FUNCTION_BLOCK FB_FanucRobot_Basic IMPLEMENTS IBasicElement
VAR_INPUT
    Estop  : BOOL; // PLC ->send to Robot E-Stop
    OpMode : E_FanucRobotOpMode := RSR01; // Select Fanuc robot prog RSR1~RSR3
    Start  : BOOL;
    Reset  : BOOL; // Reset Fanuc Robot prog
    Hold   : BOOL; // PLC - > Robot send hold command
	ManualCtrl : REFERENCE TO ST_Manual_FanucRobot;
END_VAR

VAR_OUTPUT
    qEnable       : BOOL;
    qFault        : BOOL;
    E_Stop_Output : BOOL; // Touch pannel's E-Stop has been trig;
    Halt          : BOOL; // True : Robot in helt state.
    Error         : BOOL; // True : Robot has error
    ErrorID       : UDINT; // Error ID output
	ErrMsg 		  : T_MaxString;	  
END_VAR

VAR
    // Slot1
    _rawIn_UI AT %I*  : ARRAY[0..3] OF BYTE; // UI : Fanuc robot default input rawdate
    _rawOut_UO AT %Q* : ARRAY[0..3] OF BYTE; // UO : Fanuc robot default output rawdate
    // Slot2
    _rawIn_DI AT %I*           : ARRAY[0..31] OF BYTE; // DI : user define input rawdate
    _rawOut_DO AT %Q*          : ARRAY[0..31] OF BYTE; // DO : user define output rawdate
    _EIPConnectionState AT %I* : UINT; // EIP connection State (EL6652 to Fanuc Robot)
    _FanucEIPState AT %I*      : UINT; // EIP module links to FanucRobot state
    _UI1                       : ST_FanucUI1; // Fanuc Robot default Input
    _UO1                       : ST_FanucUO1; // Fanuc Robot default Output
    _DO1                       : ST_Fanuc_WarehouseHandshake; // Fanuc robot program's handshake for clampA warehouse pick / place box
    _DO2                       : ST_Fanuc_WarehouseHandshake; // Fanuc robot program's handshake for clampB warehouse pick / place box
    _DO3                       : ST_Fanuc_AbsMove; // Fanuc robot program's handshake for clampA to target area pick / place box
    _DO4                       : ST_Fanuc_AbsMove; // Fanuc robot program's handshake for clampB to target area pick / place box
    _DO5                       : ST_Fanuc_GeneralCommand; // Fanuc robot program's handshake for general control
    _DO6                       : ST_ReadWriteParaCmd; // Fanuc robot Read/Write parameter command 
    _DO7                       : INT; // Write process X position offset
    _DO8                       : INT; // Write process Y position offset
    _DO9                       : INT; // Write process Z position offset
    _DO10                      : INT; // Write process W position offset
    _DO11                      : INT; // Write process P position offset
    _DO12                      : INT; // Write process R position offset
    _Do13                      : INT; // Write process Area index
    _Do14                      : INT; // Write process Address index
    _Do15                      : INT; // Write process Layer index
    _DO16                      : INT; // Write process Slide index
    _DO17                      : ST_CCD_ZoneUse; // Set Robot use ccd or not.
    _DI1                       : ST_Fanuc_Status; // Fanuc robot program's handshake for process status
    _DI2                       : INT; // Readprocess X position offset
    _DI3                       : INT; // Read process Y position offset
    _DI4                       : INT; // Read process Z position offset
    _DI5                       : INT; // Read process W position offset
    _DI6                       : INT; // Read process P position offset
    _DI7                       : INT; // Read process R position offset
    _DI8                       : INT; // Read process Area index
    _DI9                       : INT; // Read process Address index
    _DI10                      : INT; // Read Process Layer index
    _DI11                      : INT; // Read Process Slide index
    _DI12                      : ST_ReadWriteParaStatus; // Read/Write process Status
    _VelocityCommand           : ST_IntToBool; // Robot coordenate velocity
    // Prog inside
    eState               : E_MethodStatus_Basic;
    uiRobotExecutingStep : UINT;
    uiRobotResettingStep : UINT;
    _Error               : BOOL;
    _Abort               : BOOL;
    TON_Restart_delay    : TON;
    TON_Reset_delay      : TON;
    Rtrig_RebootRobot    : R_TRIG;
    //fbReadSingleOffsetData  : FB_ReadSingleOffsetData;
    //fbWriteSingleOffsetData : FB_WriteSingleOffsetData;
    _Status               : T_MaxString;
    _eOpMode              : E_FanucRobotOpMode;
    _ModeChanging         : BOOL;
    _Completed            : BOOL;
    _ModeChanged          : BOOL;
    _uiRSR01_Step         : UINT;
    _uiRSR02_Step         : UINT;
    _uiRSR03_Step         : UINT;
    _RetryCount           : INT := 0;
    Ton_SetProgTimeOut    : TON; // This timer is used to counting the time to switch FanucRobot prog over range.
    _RSR1_Ready           : BOOL; // Fanuc Robot running in RSR1 prog, allow to Warehouse or AbsMove command.
    _RSR2_Completed       : BOOL; // Fanuc Robot finished the homing prog.
    _RSR3_Ready           : BOOL; // Fanuc Robot ready to work.
    TON_ResetFixDelay     : TON;
    Ton_RSR_SwitchDelay   : TON; // This timer is used to counting the time to switch rsr prog
    ErrorCode             : ST_IntToBool; // This value is which read from fanuc robot.
    Ton_START_SwitchDelay : TON; // This timer is used to counting the time to switch Start signal, Fanuc process need on 0.3s and off
END_VAR

VAR CONSTANT
    RetryMaxTimes   : INT  := 3;
    tSwitchProgTime : TIME := T#1S;
    tResetFixTime   : TIME := T#0.3S;
END_VAR

// Active base units.
A00_BaseUnit();
// Active mode controller
A10_ModeControl();
// Active state controller
A20_ErrorHandle();

Update();

ACTION A00_BaseUnit:
Ton_SetProgTimeOut(PT := tSwitchProgTime);
TON_Restart_delay(PT := T#1S); // Fanuc Robot need IMSTP on over 1s
TON_Reset_delay(PT := T#1S);
TON_ResetFixDelay(PT := tResetFixTime);
Ton_RSR_SwitchDelay(PT := T#0.3S);
Ton_START_SwitchDelay(PT := T#0.4S); // Fanuc Robot need on 0.3s and then set off
E_Stop_Output := _DI12.E_Stop;
END_ACTION

ACTION A10_ModeControl:
CASE _eOpMode OF
	E_FanucRobotOpMode.RSR01:
		M_ControlRSR01(bCompleted=> _Completed, ModeChanging=> _ModeChanging, ModeChanged=> _ModeChanged);
	E_FanucRobotOpMode.RSR02:
		M_ControlRSR02(bCompleted=> _Completed, ModeChanging=> _ModeChanging, ModeChanged=> _ModeChanged);
END_CASE
END_ACTION

ACTION A20_ErrorHandle:
ErrMsg := _Status;
END_ACTION

ACTION A20_StateControl:
TON_Restart_delay(PT := T#0.5S);
TON_Reset_delay(PT:=T#0.5S);
CASE eState OF
    E_MethodStatus_Basic.STATE_DORMANT:
        Enable(FALSE);
        M_Reset(FALSE);
        uiRobotExecutingStep := 0;
        uiRobotResettingStep := 0;

		IF _eOpMode = RSR01 OR _eOpMode = RSR02 OR _eOpMode = RSR03 THEN
			eState := E_MethodStatus_Basic.STATE_EXECUTING;
		END_IF
    E_MethodStatus_Basic.STATE_EXECUTING:
        CASE uiRobotExecutingStep OF
            0:
                Enable(iTrigger := TRUE);
                M_Reset(iTrigger := TRUE);
				TON_Reset_delay.in := TRUE;
                IF TON_Reset_delay.Q THEN
                    uiRobotExecutingStep := 100;
                END_IF
            100:
                M_Reset(iTrigger := FALSE);
				TON_Reset_delay.IN := FALSE;
                IF _UO1.UO01_CmdEnabled AND _UO1.UO02_SystemReady THEN
					_VelocityCommand.nInt := 1;
                    uiRobotExecutingStep := 200;
                END_IF
            200:
				// Clear Fanuc robot's action
				GVL_ADS.AutoMode_WarehouseMotoWithRobotMove.HandShake.Execute := FALSE;
				GVL_ADS.AutoMode_RobotAbsMove.HandShake.Execute := FALSE;
				_DO1.bExecute := FALSE; // Warehouse with robot clampA
				_DO2.bExecute := FALSE; // Warehouse with robot clampB
				_DO3.bExecute := FALSE; // AbsMove with robot clampA
				_DO4.bExecute := FALSE; // AbsMove with robot clampB
				uiRobotExecutingStep := 250;
			300:
				// Switch RSR3 and read all of offset data
				GVL_ADS.FanucRobot_ReadAllOffsetData.Command.Execute := TRUE;
				IF GVL_ADS.FanucRobot_ReadAllOffsetData.Status.Done THEN
					uiRobotExecutingStep := 400;
				ELSIF GVL_ADS.FanucRobot_ReadAllOffsetData.Status.Error THEN
					_Error := TRUE;
					_Status := 'Read All offset data failue';
				END_IF
			400:
                _UI1.UI09_RSR1 := TRUE;

                IF _UO1.UO11_ACK1 THEN
                    uiRobotExecutingStep := 500;
                END_IF
            500:
                _UI1.UI09_RSR1       := FALSE;
				_VelocityCommand.nInt := 30;
                uiRobotExecutingStep := 600;
            600: // Wait command
				_DO5.ClampA_Close :=  GVL_ADS.FanucRobot_General.Command.ClampA_Close;
				_DO5.ClampA_Open := GVL_ADS.FanucRobot_General.Command.ClampA_Open;
				_DO5.ClampB_Close := GVL_ADS.FanucRobot_General.Command.ClampB_Close;
				_DO5.ClampB_Open := GVL_ADS.FanucRobot_General.Command.ClampB_Open;
				_DO6.ByPassClampSensor := GVL_ADS.FanucRobot_General.Command.ByPassClampSensor;
				GVL_ADS.FanucRobot_General.Status.ClampA_Open := _DI1.ClampA_Open;
				GVL_ADS.FanucRobot_General.Status.ClampA_Sensor := _DI1.ClampA_Sensor;
				GVL_ADS.FanucRobot_General.Status.ClampB_Open := _DI1.ClampB_Open ;
				GVL_ADS.FanucRobot_General.Status.ClampB_Sensor := _DI1.ClampB_Sensor;
				_VelocityCommand.nInt := GVL_ADS.FanucRobot_General.Command.RobotVelocity;
        END_CASE

        IF (*qFault OR *)_Error THEN
            //Soft E-Stop will cause Fault error
            eState := E_MethodStatus_Basic.STATE_ERROR;
        ELSIF _Abort THEN
            eState := E_MethodStatus_Basic.STATE_ABORTING;
		ELSIF Estop THEN
			eState := E_MethodStatus_Basic.STATE_ABORTING;
        END_IF
    E_MethodStatus_Basic.STATE_DONE:
        ;
    E_MethodStatus_Basic.STATE_ABORTING:
	;
//        Hold();

        IF _UO1.UO04_PrgPaused THEN
            eState := E_MethodStatus_Basic.STATE_Aborted;
        END_IF
    E_MethodStatus_Basic.STATE_Aborted:
        IF _UI1.UI05_FaultReset OR GVL.Reset THEN
            eState := E_MethodStatus_Basic.STATE_RESETTING;
        END_IF
    E_MethodStatus_Basic.STATE_ERROR:
        IF _UI1.UI05_FaultReset THEN
            eState := E_MethodStatus_Basic.STATE_RESETTING;
        END_IF
    E_MethodStatus_Basic.STATE_RESETTING:
        CASE uiRobotResettingStep OF
            0:
                IF NOT _UO1.UO06_Fault THEN
                    IF NOT _UO1.UO04_PrgPaused THEN
                        uiRobotResettingStep := 1000;
                    ELSE
                        uiRobotResettingStep := 2000;
                    END_IF
                ELSE
                    uiRobotResettingStep := 1000;
                END_IF
            1000:
                M_Reset(TRUE);
				TON_Reset_delay.in := TRUE;
				IF TON_Reset_delay.Q THEN
                	uiRobotResettingStep := 1010;
				END_IF
            1010:
				TON_Reset_delay.IN :=FALSE;
                M_Reset(FALSE);
                uiRobotResettingStep := 9000;
            2000:
                _UI1.UI02_Hold       := TRUE;
                TON_Restart_delay.IN := TRUE; // TimeCount start

                IF TON_Restart_delay.Q THEN
                    uiRobotResettingStep := 2100;
                END_IF
            2100:
                TON_Restart_delay.IN := FALSE;
                _UI1.UI06_Start      := TRUE;
                uiRobotResettingStep := 9000;
            9000:
                IF NOT qFault THEN
                    eState := E_MethodStatus_Basic.STATE_DORMANT;
                END_IF
        END_CASE
END_CASE
Rtrig_RebootRobot(CLK:= GVL.MachineReset.AllReset);
IF Rtrig_RebootRobot.Q	AND qFault THEN
	ReBoot();
END_IF
END_ACTION

PROPERTY AbsMoveClampA_Handshake : ST_Fanuc_AbsMove
GET
AbsMoveClampA_Handshake := _DO3;
END_GET
SET
// Outside -> FB 
_DO3 := AbsMoveClampA_Handshake;
END_SET
END_PROPERTY

PROPERTY AbsMoveClampB_Handshake : ST_Fanuc_AbsMove
GET
AbsMoveClampB_Handshake := _DO4;
END_GET
SET
// Outside -> FB 
_DO4 := AbsMoveClampB_Handshake;
END_SET
END_PROPERTY

PROPERTY Bzone_AllowWork : Bool
GET
Bzone_AllowWork := THIS^._DO6.Bzone_AllowWork;
END_GET
SET
 THIS^._DO6.Bzone_AllowWork :=Bzone_AllowWork ;
END_SET
END_PROPERTY

PROPERTY BZoneInWork : Bool
GET
BZoneInWork := THIS^._DI12.BzoneInWork;
END_GET
END_PROPERTY

PROPERTY Command : ST_FanucUO1
GET
Command := _UO1;
END_GET
SET
_UO1 := Command;
END_SET
END_PROPERTY

METHOD Enable : BOOL
VAR_INPUT
iTrigger:BOOL;
END_VAR
VAR
	_RobotEnable:BOOL;
END_VAR
_RobotEnable:=iTrigger (*AND NOT Fault()*);

_UI1.UI01_IMSP:=_RobotEnable;
_UI1.UI02_Hold:=_RobotEnable;
_UI1.UI03_SFSP:=_RobotEnable;
_UI1.UI08_Enable:=_RobotEnable;
END_METHOD

METHOD EStop
VAR_INPUT
END_VAR
_UI1.UI03_SFSP:=FALSE;
END_METHOD

PROPERTY FanucRobot_MotionStatus : ST_Fanuc_Status
GET
FanucRobot_MotionStatus := _DI1;
END_GET
END_PROPERTY

METHOD Fault : BOOL
VAR_INPUT
END_VAR
VAR_INST
	bConectionError : BOOL;
END_VAR
bConectionError := (_EIPConnectionState <>0) OR (_FanucEIPState <> 0);
Fault:=_UO1.UO06_Fault OR _UO1.UO09_BattAlarm OR _DI1.Error OR bConectionError OR _UO1.UO08_TPEnabled;
END_METHOD

METHOD GetModelState
VAR_INPUT
END_VAR
VAR_OUTPUT
    xDone : BOOL;
    xBusy : BOOL;
    xError : BOOL;
    xAborted : BOOL;
    iErrorID : UDINT;
	UniqueErrorCode : STRING;
END_VAR
xError := Error;
iErrorID := INT_TO_UDINT(ErrorCode.nInt);
END_METHOD

METHOD GetName : STRING
VAR_INPUT
END_VAR
GetName := 'Fanuc Robot';
END_METHOD

METHOD Hold
VAR_INPUT
END_VAR
_UI1.UI02_Hold:=FALSE;
END_METHOD

PROPERTY Homed : Bool
GET
Homed := _RSR2_Completed OR _UO1.UO07_AtPerch;
END_GET
END_PROPERTY

PROPERTY LayerIndex : INT
SET
_Do15 := LayerIndex;
END_SET
END_PROPERTY

METHOD M_ActiveRSR01
VAR_INPUT
END_VAR
VAR_OUTPUT
	bCompleted : BOOL;
END_VAR
CASE eState OF
    E_MethodStatus_Basic.STATE_DORMANT:
        Enable(FALSE);
        M_Reset(FALSE);
        _uiRSR01_Step        := 0;
        uiRobotExecutingStep := 0;
        uiRobotResettingStep := 0;
        _RSR1_Ready          := FALSE;
        _RSR2_Completed      := FALSE;
        _RSR3_Ready          := FALSE;
        TON_Reset_delay.IN   := FALSE;
        _RSR1_Ready          := FALSE;

        IF _eOpMode = RSR01 OR _eOpMode = RSR02 OR _eOpMode = RSR03 THEN
            eState := E_MethodStatus_Basic.STATE_EXECUTING;
        END_IF
    E_MethodStatus_Basic.STATE_EXECUTING:
        CASE uiRobotExecutingStep OF
            0:
                Enable(iTrigger := TRUE);
                TON_Restart_delay.IN := TRUE;

                IF TON_Restart_delay.Q THEN
                    uiRobotExecutingStep := 10;
                END_IF
            10:
                TON_Restart_delay.IN := FALSE;
                M_Reset(iTrigger := TRUE);
                _UI1.UI04_CycleStop  := TRUE;
                TON_ResetFixDelay.IN := TRUE;

                IF TON_ResetFixDelay.Q THEN
                    uiRobotExecutingStep := 100;
                END_IF
            100:
                TON_ResetFixDelay.IN := FALSE;
                TON_Reset_delay.in   := TRUE;
                M_Reset(iTrigger := FALSE);
                _UI1.UI04_CycleStop := FALSE;

                IF TON_Reset_delay.Q THEN
                    IF _UO1.UO01_CmdEnabled AND _UO1.UO02_SystemReady THEN
                        _Error                := FALSE;
						Enable(iTrigger := TRUE); // 20250428 Albert
                        _VelocityCommand.nInt := 1;
                        uiRobotExecutingStep  := 200;
                    ELSIF Error THEN
                        eState := E_MethodStatus_Basic.STATE_ERROR;
                    END_IF
                END_IF
            200:
                // Clear Fanuc robot's action
                TON_Reset_delay.IN                                            := FALSE;
                GVL_ADS.AutoMode_WarehouseMotoWithRobotMove.HandShake.Execute := FALSE;
                GVL_ADS.AutoMode_RobotAbsMove.HandShake.Execute               := FALSE;
                _DO1.bExecute                                                 := FALSE; // Warehouse with robot clampA
                _DO2.bExecute                                                 := FALSE; // Warehouse with robot clampB
                _DO3.bExecute                                                 := FALSE; // AbsMove with robot clampA
                _DO4.bExecute                                                 := FALSE; // AbsMove with robot clampB
                uiRobotExecutingStep                                          := 300;
            300:
                // Active RSR1
                _UI1.UI09_RSR1         := TRUE;
                Ton_SetProgTimeOut.IN  := TRUE; // Switch to RSR1 start.
                Ton_RSR_SwitchDelay.IN := TRUE;

                IF _UO1.UO11_ACK1 THEN
                    uiRobotExecutingStep := 400;
                ELSIF Error OR Ton_SetProgTimeOut.Q THEN
                    _Error  := TRUE;
                    _Status := 'RSR1 has error when RSR1 active.';
                END_IF
            400:
                // Close RSR1 command
                Ton_SetProgTimeOut.IN := FALSE; // Switch to RSR1 close.

                IF Ton_RSR_SwitchDelay.Q THEN
                    _UI1.UI09_RSR1       := FALSE;
                    uiRobotExecutingStep := 500;
                END_IF
            500:
                // Allow Robot auto / manual job
                IF (GVL_ADS.AutoMode_RobotAbsMove.HandShake.Busy OR GVL_ADS.AutoMode_RobotAbsMove.HandShake.Done) AND
                    (GVL_ADS.AutoMode_WarehouseMotoWithRobotMove.HandShake.Busy OR GVL_ADS.AutoMode_WarehouseMotoWithRobotMove.HandShake.Done) (*AND
                    (GVL_ADS.ADS_MotoCalibrationData.WDataCore.HandShake.Busy OR GVL_ADS.ADS_MotoCalibrationData.WDataCore.HandShake.Done) AND
                    (GVL_ADS.ADS_MotoCalibrationData.AbslutCore.HandShake.Busy OR GVL_ADS.ADS_MotoCalibrationData.AbslutCore.HandShake.Done)*)
                    THEN
                    bCompleted := FALSE;
                ELSE
                    bCompleted := TRUE;
                END_IF
				_Status := 'Robot in Executing State';		//edit by min 20250913   
				M_ManualService();
                //_VelocityCommand.nInt                           := GVL_ADS.FanucRobot_General.Command.RobotVelocity;
                _RSR1_Ready                                     := TRUE;

                IF _DI1.Error THEN
                    _Abort := TRUE;
                END_IF
        END_CASE

        IF _Abort THEN
            eState := E_MethodStatus_Basic.STATE_ABORTING;
        ELSIF Hold THEN
            eState := E_MethodStatus_Basic.STATE_Holding;
		ELSIF _UO1.UO06_Fault THEN
	        //_Abort := TRUE;

//			_Error  := TRUE;
//			_Status := 'Robot has fatal alarm';
//			eState  := E_MethodStatus_Basic.STATE_ERROR;
        END_IF
    E_MethodStatus_Basic.STATE_DONE:
        ;
    E_MethodStatus_Basic.STATE_ABORTING:
        eState := E_MethodStatus_Basic.STATE_ERROR;
    E_MethodStatus_Basic.STATE_Aborted:
        ;
    E_MethodStatus_Basic.STATE_ERROR:
        Enable(iTrigger := FALSE);
        _RSR1_Ready := FALSE;

        IF reset THEN
            eState := E_MethodStatus_Basic.STATE_RESETTING;
        END_IF

        IF NOT Estop AND NOT Error THEN
            eState := E_MethodStatus_Basic.STATE_RESETTING;
        END_IF
    E_MethodStatus_Basic.STATE_RESETTING:
		CASE uiRobotResettingStep OF
			0 : 
				_Error                   := FALSE;
				_Abort := false;
				_Status                  := '';
				M_ResetAllCommand();
				Ton_START_SwitchDelay.IN := FALSE;
				TON_Restart_delay.IN := FALSE;
				uiRobotResettingStep := 10;
			10:
				M_Reset(iTrigger :=TRUE);
				TON_Restart_delay.IN := TRUE;
				IF TON_Restart_delay.Q THEN
					M_EnableWith4Input(TRUE	,TRUE,TRUE,FALSE);
					uiRobotResettingStep := 20;
				END_IF
			20:
				TON_Restart_delay.IN := FALSE;
				M_Reset(iTrigger :=FALSE);
        		//Enable(iTrigger := TRUE);
				IF NOT  _UO1.UO06_Fault THEN
					M_EnableWith4Input(TRUE	,TRUE,TRUE,FALSE);
					uiRobotResettingStep := 50;
				END_IF
				IF reset THEN
					uiRobotResettingStep := 0;
				END_IF
			30 :
				M_Reset(iTrigger :=TRUE);
				uiRobotResettingStep := 40;
			40:
				M_Reset(iTrigger :=FALSE);
				uiRobotResettingStep := 50;
			50:
				IF reset THEN
					uiRobotResettingStep := 0;
				END_IF
				IF NOT Error THEN
					eState := E_MethodStatus_Basic.STATE_DORMANT;
				END_IF
		END_CASE
    E_MethodStatus_Basic.STATE_Holding:
        _UI1.UI02_Hold := FALSE;

        IF _UO1.UO04_PrgPaused AND NOT _UO1.UO03_PrgRunning THEN
            Halt    := TRUE;
            _Status := 'Robot in Halt State';
            eState  := E_MethodStatus_Basic.STATE_Held;
        END_IF
		IF reset THEN
			eState         := E_MethodStatus_Basic.STATE_ERROR;
		END_IF
    E_MethodStatus_Basic.STATE_Held:
		Ton_START_SwitchDelay.IN := FALSE;
        IF reset AND NOT Hold THEN
			//M_Reset(iTrigger:=TRUE);		//edit by min , if need resume robot motion dont set robot UI04 cyclestop
			_UI1.UI05_FaultReset:=TRUE;
            Halt := FALSE;
		ELSE
			M_Reset(iTrigger :=FALSE);
        END_IF

        IF NOT Halt AND Start THEN
            _UI1.UI02_Hold := TRUE;
            eState         := E_MethodStatus_Basic.STATE_UnHold;
        END_IF
    E_MethodStatus_Basic.STATE_UnHold:
        Ton_START_SwitchDelay.IN := TRUE;
		 _UI1.UI09_RSR1         := TRUE;
        _UI1.UI06_Start          := NOT Ton_START_SwitchDelay.Q;
		
        IF NOT _UO1.UO04_PrgPaused AND _UO1.UO03_PrgRunning AND NOT _UI1.UI06_Start THEN
            Ton_START_SwitchDelay.IN := FALSE;
			 _UI1.UI09_RSR1         := FALSE;
            eState                   := E_MethodStatus_Basic.STATE_EXECUTING;
        END_IF
END_CASE

IF Estop THEN
   // _Error  := TRUE;
    _Status := 'EStop has been trigged.';
	eState  := E_MethodStatus_Basic.STATE_ERROR;
ELSIF _UO1.UO08_TPEnabled THEN
    _Error  := TRUE;
    _Status := 'TP has got contol';
	eState  := E_MethodStatus_Basic.STATE_ERROR;
ELSIF _UO1.UO09_BattAlarm THEN
    _Error  := TRUE;
    _Status := 'Robot has Battary alarm';
	eState  := E_MethodStatus_Basic.STATE_ERROR;
END_IF
END_METHOD

METHOD M_ActiveRSR02
VAR_INPUT
END_VAR
VAR_OUTPUT
	bCompleted : BOOL;
END_VAR
CASE eState OF
	E_MethodStatus_Basic.STATE_DORMANT:
        Enable(FALSE);
        M_Reset(FALSE);
        _uiRSR01_Step := 0;
		uiRobotExecutingStep := 0;
        uiRobotResettingStep := 0;
		_RSR1_Ready := FALSE;
		_RSR2_Completed := FALSE;
		_RSR3_Ready:=FALSE;
		TON_Reset_delay.IN := FALSE;
		IF _eOpMode = RSR01 OR _eOpMode = RSR02 OR _eOpMode = RSR03 THEN
			eState := E_MethodStatus_Basic.STATE_EXECUTING;
		END_IF
	E_MethodStatus_Basic.STATE_EXECUTING:
		CASE uiRobotExecutingStep OF
			0:
                Enable(iTrigger := TRUE);
				TON_Restart_delay.IN := TRUE;
				IF TON_Restart_delay.Q THEN
					uiRobotExecutingStep := 10;
				END_IF
			10:
				TON_Restart_delay.IN := FALSE;
                M_Reset(iTrigger := TRUE);
				TON_ResetFixDelay.in := TRUE;
				_UI1.UI04_CycleStop := TRUE;
				IF TON_ResetFixDelay.Q THEN
	                uiRobotExecutingStep := 100;
				END_IF
			100:
				TON_ResetFixDelay.in := FALSE;
				TON_Reset_delay.in := TRUE;
                M_Reset(iTrigger := FALSE);
				_UI1.UI04_CycleStop := FALSE;
				IF TON_Reset_delay.Q THEN
					IF _UO1.UO01_CmdEnabled AND _UO1.UO02_SystemReady THEN
						_VelocityCommand.nInt := 1;
						uiRobotExecutingStep := 200;
					ELSIF Error THEN
						eState := E_MethodStatus_Basic.STATE_ERROR;
					END_IF
				END_IF
			200:
				// Clear Fanuc robot's action
				GVL_ADS.AutoMode_WarehouseMotoWithRobotMove.HandShake.Execute := FALSE;
				GVL_ADS.AutoMode_RobotAbsMove.HandShake.Execute := FALSE;
				_DO1.bExecute := FALSE;
				_DO2.bExecute := FALSE;
				_DO3.bExecute := FALSE;
				_DO4.bExecute := FALSE;
				uiRobotExecutingStep := 300;
			300:
				// Switch RSR02
				_UI1.UI10_RSR2 := TRUE;
		
				IF _UO1.UO12_ACK2 THEN
					uiRobotExecutingStep := 400;
				END_IF
			400:
				_UI1.UI10_RSR2 := FALSE;
				IF (_DI1.Done OR _UO1.UO07_AtPerch )  
				THEN
					uiRobotExecutingStep := 9900;
				END_IF
			9900:
				eState := E_MethodStatus_Basic.STATE_DONE;
		END_CASE
	E_MethodStatus_Basic.STATE_DONE:
		_RSR2_Completed := TRUE;
		bCompleted := TRUE;
	E_MethodStatus_Basic.STATE_ABORTING:
		;
	E_MethodStatus_Basic.STATE_Aborted:
		;
	E_MethodStatus_Basic.STATE_ERROR:
		Enable(iTrigger := FALSE);
		IF reset THEN
			eState := E_MethodStatus_Basic.STATE_RESETTING;
		END_IF
		IF NOT Estop AND NOT Error THEN
			eState := E_MethodStatus_Basic.STATE_RESETTING;
		END_IF
	E_MethodStatus_Basic.STATE_RESETTING:
		eState := E_MethodStatus_Basic.STATE_DORMANT;
END_CASE
IF Estop OR _UO1.UO08_TPEnabled THEN
	eState := E_MethodStatus_Basic.STATE_ERROR;
	_Error := TRUE;
	_Status := 'EStop has been trigged.';
END_IF
END_METHOD

METHOD M_ActiveRSR03
VAR_INPUT
END_VAR
VAR_OUTPUT
	bCompleted : BOOL;
END_VAR
CASE _uiRSR03_Step OF
	0:
		// Stop Prog
		_RSR1_Ready := FALSE;
		_RSR2_Completed := FALSE;
		_RSR3_Ready:=FALSE;
		_UI1.UI04_CycleStop := TRUE;
		IF NOT _UO1.UO04_PrgPaused AND NOT _UO1.UO03_PrgRunning THEN
			_uiRSR03_Step := 100;
		END_IF
	100:
		// Close cycle stop
		_UI1.UI04_CycleStop := FALSE;
		// Set current prog - RSR03
		_UI1.UI11_RSR3 := TRUE;
		IF _UO1.UO13_ACK3 THEN
			_uiRSR03_Step := 200;
		END_IF
	200:
		// Clear RSR03 command 
		_UI1.UI11_RSR3 := FALSE;
		_uiRSR03_Step := 300;
	300:
		// Allow Read / Write offset data
		IF ( GVL_ADS.FanucRobot_ReadAllOffsetData.Status.Busy  OR GVL_ADS.FanucRobot_ReadAllOffsetData.Status.Done) AND
			(GVL_ADS.FanucRobot_ReadSingleOffsetData.Status.Busy OR GVL_ADS.FanucRobot_ReadSingleOffsetData.Status.Done) AND
			(GVL_ADS.FanucRobot_WirteSingleOffsetData.Status.Busy OR GVL_ADS.FanucRobot_WirteSingleOffsetData.Status.Done ) AND
			(GVL_ADS.FanucRobot_WriteAllOffsetData.Status.Busy OR GVL_ADS.FanucRobot_WriteAllOffsetData.Status.Done) 
		THEN
			_RSR3_Ready := FALSE;
			bCompleted := FALSE;
		ELSE
			_RSR3_Ready := FALSE;
			bCompleted := TRUE;
		END_IF 
		
END_CASE

CASE eState OF
	E_MethodStatus_Basic.STATE_DORMANT:
        Enable(FALSE);
        M_Reset(FALSE);
        _uiRSR01_Step := 0;
		uiRobotExecutingStep := 0;
        uiRobotResettingStep := 0;
		_RSR1_Ready := FALSE;
		_RSR2_Completed := FALSE;
		_RSR3_Ready:=FALSE;
		TON_Reset_delay.IN := FALSE;
		IF _eOpMode = RSR01 OR _eOpMode = RSR02 OR _eOpMode = RSR03 THEN
			eState := E_MethodStatus_Basic.STATE_EXECUTING;
		END_IF
	E_MethodStatus_Basic.STATE_EXECUTING:
		CASE uiRobotExecutingStep OF
			0:
                Enable(iTrigger := TRUE);
				TON_Restart_delay.IN := TRUE;
				IF TON_Restart_delay.Q THEN
					uiRobotExecutingStep := 10;
				END_IF
			10:
				TON_Restart_delay.IN := FALSE;
                M_Reset(iTrigger := TRUE);
				_UI1.UI04_CycleStop := TRUE;
				TON_ResetFixDelay.IN := TRUE;
				IF TON_ResetFixDelay.Q THEN
                	uiRobotExecutingStep := 100;
				END_IF
			100:
				TON_ResetFixDelay.IN := FALSE;
				TON_Reset_delay.in := TRUE;
                M_Reset(iTrigger := FALSE);
				_UI1.UI04_CycleStop := FALSE;
				IF TON_Reset_delay.Q THEN
					IF _UO1.UO01_CmdEnabled AND _UO1.UO02_SystemReady THEN
						_VelocityCommand.nInt := 1;
						uiRobotExecutingStep := 200;
					ELSIF Error THEN
						eState := E_MethodStatus_Basic.STATE_ERROR;
					END_IF
				END_IF
			200:
				// Clear Fanuc robot's action
				TON_Reset_delay.IN := FALSE;
				GVL_ADS.AutoMode_WarehouseMotoWithRobotMove.HandShake.Execute := FALSE;
				GVL_ADS.AutoMode_RobotAbsMove.HandShake.Execute := FALSE;
				_DO1.bExecute := FALSE; // Warehouse with robot clampA
				_DO2.bExecute := FALSE; // Warehouse with robot clampB
				_DO3.bExecute := FALSE; // AbsMove with robot clampA
				_DO4.bExecute := FALSE; // AbsMove with robot clampB
				uiRobotExecutingStep := 300;
			300:
				// Active RSR1
                _UI1.UI11_RSR3 := TRUE;
                IF _UO1.UO13_ACK3 THEN
                    uiRobotExecutingStep := 400;
				ELSIF Error THEN
					_Error := TRUE;
					_Status:='RSR3 has error when RSR3 active.';
                END_IF
			400:
				// Allow Read / Write offset data
				IF ( GVL_ADS.FanucRobot_ReadAllOffsetData.Status.Busy  OR GVL_ADS.FanucRobot_ReadAllOffsetData.Status.Done) AND
					(GVL_ADS.FanucRobot_ReadSingleOffsetData.Status.Busy OR GVL_ADS.FanucRobot_ReadSingleOffsetData.Status.Done) AND
					(GVL_ADS.FanucRobot_WirteSingleOffsetData.Status.Busy OR GVL_ADS.FanucRobot_WirteSingleOffsetData.Status.Done ) AND
					(GVL_ADS.FanucRobot_WriteAllOffsetData.Status.Busy OR GVL_ADS.FanucRobot_WriteAllOffsetData.Status.Done) 
				THEN
					_RSR3_Ready := FALSE;
					bCompleted := FALSE;
				ELSE
					_RSR3_Ready := FALSE;
					bCompleted := TRUE;
				END_IF 
		END_CASE
	E_MethodStatus_Basic.STATE_DONE:
		;
	E_MethodStatus_Basic.STATE_ABORTING:
		;
	E_MethodStatus_Basic.STATE_Aborted:
		;
	E_MethodStatus_Basic.STATE_ERROR:
		Enable(iTrigger := FALSE);
		IF Reset THEN
			eState := E_MethodStatus_Basic.STATE_RESETTING;
		END_IF
		IF  Estop AND NOT Error THEN
			eState := E_MethodStatus_Basic.STATE_RESETTING;
		END_IF
	E_MethodStatus_Basic.STATE_RESETTING:
		eState := E_MethodStatus_Basic.STATE_DORMANT;
END_CASE

IF Estop OR _UO1.UO08_TPEnabled THEN
	eState := E_MethodStatus_Basic.STATE_ERROR;
	_Error := TRUE;
	_Status := 'EStop has been trigged.';
END_IF
END_METHOD

METHOD M_ClearState : BOOL;
VAR_INPUT
END_VAR

eState := E_MethodStatus_Basic.STATE_DORMANT;
uiRobotExecutingStep := 0;
uiRobotResettingStep := 0;
M_ClearState := TRUE;
END_METHOD

METHOD M_ControlRSR01
VAR_INPUT
END_VAR
VAR_OUTPUT
	bCompleted : BOOL;
	ModeChanging : BOOL;
	ModeChanged : BOOL;
END_VAR
ModeChanging := FALSE;
ModeChanged := TRUE;
M_ActiveRSR01(bCompleted => bCompleted);

IF OpMode <> _eOpMode (*AND bCompleted*) THEN
    _uiRSR01_Step := 0;
    eState := E_MethodStatus_Basic.STATE_DORMANT;
    _eOpMode := OpMode;
END_IF
END_METHOD

METHOD M_ControlRSR02
VAR_INPUT
END_VAR
VAR_OUTPUT
    bCompleted : BOOL;
    ModeChanging : BOOL;
    ModeChanged : BOOL;
END_VAR
ModeChanging := FALSE;
ModeChanged := TRUE;
M_ActiveRSR02(bCompleted => bCompleted);

IF OpMode <> _eOpMode AND bCompleted THEN
    _uiRSR02_Step := 0;
    eState := E_MethodStatus_Basic.STATE_DORMANT;
    _eOpMode := OpMode;
END_IF
END_METHOD

METHOD M_ControlRSR03

VAR_INPUT
END_VAR
VAR_OUTPUT
    bCompleted : BOOL;
    ModeChanging : BOOL;
    ModeChanged : BOOL;
END_VAR
ModeChanging := FALSE;
ModeChanged := TRUE;
M_ActiveRSR03(bCompleted => bCompleted);

IF OpMode <> _eOpMode AND bCompleted THEN
	_uiRSR03_Step := 0;
	eState := E_MethodStatus_Basic.STATE_DORMANT;
	_eOpMode := OpMode;
END_IF
END_METHOD

METHOD PRIVATE M_EnableWith4Input : BOOL
VAR_INPUT
	IMSP : BOOL;
	Hold : BOOL;
	SFSP : BOOL;
	Enable : BOOL;
END_VAR
_UI1.UI01_IMSP:=IMSP;
_UI1.UI02_Hold:=Hold;
_UI1.UI03_SFSP:=SFSP;
_UI1.UI08_Enable:=Enable;
END_METHOD

METHOD M_GetErrorCode : Int
VAR_INPUT
END_VAR
ErrorCode.BitList.Bit0 := _DI1.ErrorID_01;
ErrorCode.BitList.Bit1 := _DI1.ErrorID_02;
ErrorCode.BitList.Bit2 := _DI1.ErrorID_03;
ErrorCode.BitList.Bit3 := _DI1.ErrorID_04;
ErrorCode.BitList.Bit4 := _DI1.ErrorID_05;
ErrorCode.BitList.Bit5 := _DI1.ErrorID_06;
ErrorCode.BitList.Bit6 := _DI1.ErrorID_07;
ErrorCode.BitList.Bit7 := _DI1.ErrorID_08;		
//ErrorCode.BitList.Bit8 := _DI1.ErrorID_09;
//ErrorCode.BitList.Bit9 := _DI1.ErrorID_10;
M_GetErrorCode := ErrorCode.nInt;
END_METHOD

METHOD M_Kawasaki_API
VAR_INPUT
	WarehouseClampA_Handshake : UINT;
	WarehouseClampB_Handshake : UINT;
	AbsMoveClampA_Handshake : UINT;
	AbsMoveClampB_Handshake : UINT;
END_VAR
VAR_OUTPUT
	Status : UINT;
END_VAR
MEMMOVE(destAddr:=ADR(_DO1),srcAddr:=ADR(WarehouseClampA_Handshake),n:=2);
MEMMOVE(destAddr:=ADR(_DO2),srcAddr:=ADR(WarehouseClampB_Handshake),n:=2);
MEMMOVE(destAddr:=ADR(_DO3),srcAddr:=ADR(AbsMoveClampA_Handshake),n:=2);
MEMMOVE(destAddr:=ADR(_DO4),srcAddr:=ADR(AbsMoveClampB_Handshake),n:=2);
IF NOT _UO1.UO08_TPEnabled THEN
	MEMMOVE(destAddr:=ADR(Status),srcAddr:=ADR(_DI1),n:=2);
END_IF
END_METHOD

METHOD M_ManualService
VAR_INPUT
END_VAR
_DO5.ClampA_Close := ManualCtrl.ClampA_Close;
_DO5.ClampA_Open := ManualCtrl.ClampA_Open;
_DO5.ClampB_Close := ManualCtrl.ClampB_Close;
_DO5.ClampB_Open := ManualCtrl.ClampB_Open;
_DO6.ByPassClampSensor := ManualCtrl.ByPassClampSensor;
GVL_ADS.FanucRobot_General.Status.ClampA_Open := _DI1.ClampA_Open;
GVL_ADS.FanucRobot_General.Status.ClampA_Sensor := _DI1.ClampA_Sensor;
GVL_ADS.FanucRobot_General.Status.ClampB_Open := _DI1.ClampB_Open;
GVL_ADS.FanucRobot_General.Status.ClampB_Sensor := _DI1.ClampB_Sensor;
END_METHOD

METHOD M_Reset : BOOL
VAR_INPUT
	iTrigger:BOOL;
END_VAR
_UI1.UI05_FaultReset:=iTrigger;
_UI1.UI04_CycleStop:=iTrigger;
END_METHOD

METHOD M_ResetAbsMoveClampACommand : BOOL
VAR_INPUT
END_VAR
VAR
	SpareData : ST_Fanuc_AbsMove;
END_VAR
_DO3 := SpareData;

M_ResetAbsMoveClampACommand := TRUE; // Method end
END_METHOD

METHOD M_ResetAbsMoveClampBCommand : BOOL
VAR_INPUT
END_VAR
VAR
	SpareData : ST_Fanuc_AbsMove;
END_VAR
_DO4 := SpareData;

M_ResetAbsMoveClampBCommand := true; // Method end
END_METHOD

METHOD M_ResetAbsMoveCommand : BOOL
VAR_INPUT
END_VAR
// Clear AbsMove ClampA command data
M_ResetAbsMoveClampACommand();
// Clear AbsMove ClampB command data
M_ResetAbsMoveClampBCommand();

M_ResetAbsMoveCommand := TRUE; // Method end
END_METHOD

METHOD M_ResetAllCommand : BOOL
VAR_INPUT
END_VAR
// Clear WareHouse command
M_ResetWareHouseCommand();
// Clear AbsMove Command
M_ResetAbsMoveCommand();

M_ResetAllCommand := TRUE; // Method end
END_METHOD

METHOD M_ResetMoveBoxToFeedInConveyor_ClampA : BOOL
VAR_INPUT
END_VAR
VAR
	SpaceData : ST_Fanuc_AbsMove;
END_VAR
_DO3 := SpaceData;

M_ResetMoveBoxToFeedInConveyor_ClampA := TRUE; // Mehtod end
END_METHOD

METHOD M_ResetMoveBoxToFeedInConveyor_ClampB : BOOL
VAR_INPUT
END_VAR
VAR
    SpaceData : ST_Fanuc_AbsMove;
END_VAR
_DO4 := SpaceData;

M_ResetMoveBoxToFeedInConveyor_ClampB := TRUE; // Method end
END_METHOD

METHOD M_ResetMoveBoxToFeedInConveyor_ClampBoth : BOOL
VAR_INPUT
END_VAR
VAR
    SpaceData : ST_Fanuc_AbsMove;
END_VAR
_DO3 := SpaceData;
_DO4 := SpaceData;

M_ResetMoveBoxToFeedInConveyor_ClampBoth := TRUE; // Method end
END_METHOD

METHOD M_ResetMoveBoxToRoundBelt_Both : BOOL
VAR_INPUT
END_VAR
VAR
    SpaceData : ST_Fanuc_AbsMove;
END_VAR
_DO3 := SpaceData;
_DO4 := SpaceData;

M_ResetMoveBoxToRoundBelt_Both := TRUE; // Method end
END_METHOD

METHOD M_ResetPullOutConveyorPickUpBox_ClampA : BOOL
VAR_INPUT
END_VAR
VAR
	SpaceData : ST_Fanuc_AbsMove;
END_VAR
_DO3 := SpaceData;

M_ResetPullOutConveyorPickUpBox_ClampA := TRUE; // Method end
END_METHOD

METHOD M_ResetPullOutConveyorPickUpBox_ClampB : BOOL
VAR_INPUT
END_VAR
VAR
    SpaceData : ST_Fanuc_AbsMove;
END_VAR
_DO4 := SpaceData;

M_ResetPullOutConveyorPickUpBox_ClampB := true; // Method end
END_METHOD

METHOD M_ResetPullOutConveyorPickUpBox_ClampBoth : BOOL
VAR_INPUT
END_VAR
VAR
    SpaceData : ST_Fanuc_AbsMove;
END_VAR
_DO3 := SpaceData;
_DO4 := SpaceData;

M_ResetPullOutConveyorPickUpBox_ClampBoth := TRUE; // Method end
END_METHOD

METHOD PUBLIC M_ResetRobotAbsMove : BOOL
VAR_INPUT
	ResetClampA : BOOL;
	ResetClampB : BOOL;
END_VAR

VAR
	SpaceData : ST_Fanuc_AbsMove;
END_VAR
IF ResetClampA THEN
	_DO3 := SpaceData;
END_IF

IF ResetClampB THEN
	_DO4 := SpaceData;
END_IF

M_ResetRobotAbsMove:=True;
END_METHOD

METHOD M_ResetWareHouseClampACommand : BOOL
VAR_INPUT
END_VAR
VAR
	SpareData : ST_Fanuc_WarehouseHandshake;
END_VAR
_DO1 := SpareData;

M_ResetWareHouseClampACommand := TRUE; // Method end
END_METHOD

METHOD M_ResetWareHouseClampBCommand : BOOL
VAR_INPUT
END_VAR
VAR
	SpareData : ST_Fanuc_WarehouseHandshake;
END_VAR
_DO2 := SpareData;

M_ResetWareHouseClampBCommand := true; // Method end
END_METHOD

METHOD M_ResetWareHouseCommand : BOOL
VAR_INPUT
END_VAR
// Clear WareHouse ClampA command data
M_ResetWareHouseClampACommand();
// Clear WareHouse ClampB command data
M_ResetWareHouseClampBCommand();

M_ResetWareHouseCommand := TRUE; // Method end
END_METHOD

METHOD M_ResetWareHousePickUpBox_ClampA : BOOL
VAR_INPUT
END_VAR
VAR
	SpaceData :ST_Fanuc_WarehouseHandshake;
END_VAR
// Clear command
_DO1 := SpaceData;

M_ResetWareHousePickUpBox_ClampA := TRUE; // Method End
END_METHOD

METHOD M_ResetWareHousePickUpBox_ClampB : BOOL
VAR_INPUT
END_VAR
VAR
	SpaceData :ST_Fanuc_WarehouseHandshake;
END_VAR
// Clear command
_DO2 := SpaceData;

M_ResetWareHousePickUpBox_ClampB := TRUE; // Method End
END_METHOD

METHOD M_ResetWareHousePickUpBox_ClampBoth : BOOL
VAR_INPUT
END_VAR
VAR
	SpaceData :ST_Fanuc_WarehouseHandshake;
END_VAR
// Clear command
_DO1 := SpaceData;
_DO2 := SpaceData;

M_ResetWareHousePickUpBox_ClampBoth := TRUE; // Method end
END_METHOD

(* This Method is used to send command data to Fanuc Robot, only clampA is work 
*)
METHOD M_StartAbsMoveAction_ClampA : BOOL
VAR_INPUT
	TargetArea : E_RobotArea; // Select the zone where robot will going.
	TargetAddress : E_RobotAddress; // Because the address num in different zone, the number define is different. But also need >= 1, 0 = undefined
	ClampAction : E_ClampAction; // need to define the command
	BoxReady : BOOL; // Fanuc robot prog will stop at a safe position just before reaching the target location, until `AllowContinue` is set to true.
END_VAR

VAR_OUTPUT
    Error  : BOOL;
    ErrMsg : T_MaxString;
END_VAR

VAR_INST
	_Area : ST_IntToBool;
	_Address : ST_IntToBool;
END_VAR
// Set target area
_Area.nInt := TargetArea;

CASE TargetArea OF
    E_RobotArea.RoundBelt..E_RobotArea.PullOutConveyor:
        _Area.nInt := TargetArea;
ELSE
    Error  := TRUE;
    ErrMsg := 'ClampA target area out of range';
	RETURN;
END_CASE

// Set target address
_Address.nInt := TargetAddress;

CASE TargetAddress OF
    E_RobotAddress.Address01..E_RobotAddress.Address06:
        _Address.nInt := TargetAddress;
ELSE
    Error  := TRUE;
    ErrMsg := 'ClampA target address out of range';
	RETURN;
END_CASE

// Check ClampA Action is correct
CASE ClampAction OF
	E_ClampAction.PickUp:
		_DO3.bGet := TRUE;
	E_ClampAction.Place:
		_DO3.bGet := FALSE;
ELSE
	Error := TRUE;
	ErrMsg := 'ClampA Action is wrong command';
	RETURN;
END_CASE

// Send robot target area data
_DO3.nArea1 := _Area.BitList.Bit0;
_DO3.nArea2 := _Area.BitList.Bit1;
_DO3.nArea3 := _Area.BitList.Bit2;
_DO3.nArea4 := _Area.BitList.Bit3;

// Send robot target address data
_DO3.nAddress1 := _Address.BitList.Bit0;
_DO3.nAddress2 := _Address.BitList.Bit1;
_DO3.nAddress3 := _Address.BitList.Bit2;
_DO3.nAddress4 := _Address.BitList.Bit3;
_DO3.nAddress5 := _Address.BitList.Bit4;
_DO3.nAddress6 := _Address.BitList.Bit5;
_DO3.nAddress7 := _Address.BitList.Bit6;


_DO3.bExecute := NOT Error;

_DO3.bContinue := BoxReady;

M_StartAbsMoveAction_ClampA := NOT Error; // Method end
END_METHOD

(* This Method is used to send command data to Fanuc Robot, only clampB is work 
*)
METHOD M_StartAbsMoveAction_ClampB : BOOL
VAR_INPUT
    TargetArea    : E_RobotArea;    // Select the zone where robot will going.
    TargetAddress : E_RobotAddress; // Because the address num in different zone, the number define is different. But also need >= 1, 0 = undefined
    ClampAction   : E_ClampAction;  // need to define the command
    BoxReady      : BOOL;           // Fanuc robot prog will stop at a safe position just before reaching the target location, until `AllowContinue` is set to true.
END_VAR

VAR_OUTPUT
    Error  : BOOL;
    ErrMsg : T_MaxString;
END_VAR

VAR_INST
    _Area    : ST_IntToBool;
    _Address : ST_IntToBool;
END_VAR
// Set target area
_Area.nInt := TargetArea;

// Check ClampB target area is correct
CASE TargetArea OF
    E_RobotArea.RoundBelt..E_RobotArea.PullOutConveyor:
        _Area.nInt := TargetArea;
ELSE
    Error  := TRUE;
    ErrMsg := 'ClampB target area out of range';
	RETURN;
END_CASE

// Check ClampB target address is correct
CASE TargetAddress OF
	E_RobotAddress.Address01..E_RobotAddress.Address06:
		_Address.nInt := TargetAddress;
ELSE
	Error := TRUE;
	ErrMsg := 'ClampB target address is out of range';
	RETURN;
END_CASE

// Check ClampB Action is correct
CASE ClampAction OF
	E_ClampAction.PickUp:
		_DO4.bGet := TRUE;
	E_ClampAction.Place:
		_DO4.bGet := FALSE;
ELSE
	Error := TRUE;
	ErrMsg := 'ClampB Action is wrong command';
	RETURN;
END_CASE

// Send robot target area data
_DO4.nArea1 := _Area.BitList.Bit0;
_DO4.nArea2 := _Area.BitList.Bit1;
_DO4.nArea3 := _Area.BitList.Bit2;
_DO4.nArea4 := _Area.BitList.Bit3;

// Send robot target address data
_DO4.nAddress1 := _Address.BitList.Bit0;
_DO4.nAddress2 := _Address.BitList.Bit1;
_DO4.nAddress3 := _Address.BitList.Bit2;
_DO4.nAddress4 := _Address.BitList.Bit3;
_DO4.nAddress5 := _Address.BitList.Bit4;
_DO4.nAddress6 := _Address.BitList.Bit5;
_DO4.nAddress7 := _Address.BitList.Bit6;

_DO4.bExecute := NOT Error;

_DO4.bContinue := BoxReady;

M_StartAbsMoveAction_ClampB := NOT Error; // Method end
END_METHOD

METHOD M_StartAbsMoveAction_ClampBoth : BOOL
VAR_INPUT
    ClampA_TargetArea    : E_RobotArea;
    ClampA_TargetAddress : E_RobotAddress;
    ClampA_Action        : E_ClampAction;
    ClampB_TargetArea    : E_RobotArea;
    ClampB_TargetAddress : E_RobotAddress;
    ClampB_Action        : E_ClampAction;
    BoxReady_1st         : BOOL;
    BoxReady_2nd         : BOOL;
END_VAR

VAR_OUTPUT
    Error  : BOOL;
    ErrMsg : T_MaxString;
END_VAR

VAR_INST
    _ClampA_Area    : ST_IntToBool;
    _ClampB_Area    : ST_IntToBool;
    _ClampA_Address : ST_IntToBool;
    _ClampB_Address : ST_IntToBool;
END_VAR
// Set Target Area
_ClampA_Area.nInt := ClampA_TargetArea;
_ClampB_Area.nInt := ClampB_TargetArea;
// Check ClampA target area is correct
CASE ClampA_TargetArea OF
    E_RobotArea.RoundBelt..E_RobotArea.PullOutConveyor:
        _ClampA_Area.nInt := ClampA_TargetArea;
ELSE
    Error  := TRUE;
    ErrMsg := 'ClampA target area out of range';
	RETURN;
END_CASE
// Check ClampA target address is correct
CASE ClampA_TargetAddress OF
    E_RobotAddress.Address01..E_RobotAddress.Address06:
        _ClampA_Address.nInt := ClampA_TargetAddress;
ELSE
    Error  := TRUE;
    ErrMsg := 'ClampA target address out of range';
	RETURN;
END_CASE

// Check ClampA Action is correct
CASE ClampA_Action OF
	E_ClampAction.PickUp:
		_DO3.bGet := TRUE;
	E_ClampAction.Place:
		_DO3.bGet := FALSE;
ELSE
	Error := TRUE;
	ErrMsg := 'ClampA Action is wrong command';
	RETURN;
END_CASE
// Check ClampB target area is correct
CASE ClampB_TargetArea OF
    E_RobotArea.RoundBelt..E_RobotArea.PullOutConveyor:
        _ClampB_Area.nInt := ClampB_TargetArea;
ELSE
	Error := TRUE;
	ErrMsg := 'ClampB target area out of range';
	RETURN;
END_CASE

// Check ClampB target address is correct
CASE ClampB_TargetAddress OF
	E_RobotAddress.Address01..E_RobotAddress.Address06:
		_ClampB_Address.nInt := ClampB_TargetAddress;
ELSE
	Error := TRUE;
	ErrMsg := 'ClampB target address is out of range';
	RETURN;
END_CASE
// Check ClampB Action is correct
CASE ClampB_Action OF
	E_ClampAction.PickUp:
		_DO4.bGet := TRUE;
	E_ClampAction.Place:
		_DO4.bGet := FALSE;
ELSE
	Error := TRUE;
	ErrMsg := 'ClampB Action is wrong command';
	RETURN;
END_CASE

// Send robot target area data
_DO3.nArea1 := _ClampA_Area.BitList.Bit0;
_DO3.nArea2 := _ClampA_Area.BitList.Bit1;
_DO3.nArea3 := _ClampA_Area.BitList.Bit2;
_DO3.nArea4 := _ClampA_Area.BitList.Bit3;

_DO4.nArea1 := _ClampB_Area.BitList.Bit0;
_DO4.nArea2 := _ClampB_Area.BitList.Bit1;
_DO4.nArea3 := _ClampB_Area.BitList.Bit2;
_DO4.nArea4 := _ClampB_Area.BitList.Bit3;

// Send robot target address data
_DO3.nAddress1 := _ClampA_Address.BitList.Bit0;
_DO3.nAddress2 := _ClampA_Address.BitList.Bit1;
_DO3.nAddress3 := _ClampA_Address.BitList.Bit2;
_DO3.nAddress4 := _ClampA_Address.BitList.Bit3;
_DO3.nAddress5 := _ClampA_Address.BitList.Bit4;
_DO3.nAddress6 := _ClampA_Address.BitList.Bit5;
_DO3.nAddress7 := _ClampA_Address.BitList.Bit6;

_DO4.nAddress1 := _ClampB_Address.BitList.Bit0;
_DO4.nAddress2 := _ClampB_Address.BitList.Bit1;
_DO4.nAddress3 := _ClampB_Address.BitList.Bit2;
_DO4.nAddress4 := _ClampB_Address.BitList.Bit3;
_DO4.nAddress5 := _ClampB_Address.BitList.Bit4;
_DO4.nAddress6 := _ClampB_Address.BitList.Bit5;
_DO4.nAddress7 := _ClampB_Address.BitList.Bit6;

_DO3.bExecute := NOT Error;
_DO4.bExecute := NOT Error;

_DO3.bContinue := BoxReady_1st;
_DO4.bContinue := BoxReady_2nd;

M_StartAbsMoveAction_ClampBoth := NOT Error; // Method end
END_METHOD

METHOD M_StartMoveBoxToFeedInConveyor_ClampA : BOOL
VAR_INPUT
    ConveyorSlideSelect : E_FeedInEmptyBox_PlaceArea;
    DiffSizeSlideClear  : BOOL;
    SameSizeSlideClear  : BOOL;
END_VAR
VAR_INST
    _Area    : ST_IntToBool;
    _Address : ST_IntToBool;
END_VAR
// Set target area is round belt
_Area.nInt := E_RobotArea.TransmitCV;
IF ConveyorSlideSelect = E_FeedInEmptyBox_PlaceArea.DiffSizeConveyor THEN
	_Address.nInt := 1;
ELSIF ConveyorSlideSelect = E_FeedInEmptyBox_PlaceArea.SameSizeConveyor THEN
	_Address.nInt := 2;
ELSE
	// Wrong command, return
	RETURN ;
END_IF
// Send robot target area data
_DO3.nArea1 := _Area.BitList.Bit0;
_DO3.nArea2 := _Area.BitList.Bit1;
_DO3.nArea3 := _Area.BitList.Bit2;
_DO3.nArea4 := _Area.BitList.Bit3;

// Send robot target address data
_DO3.nAddress1 := _Address.BitList.Bit0;
_DO3.nAddress2 := _Address.BitList.Bit1;
_DO3.nAddress3 := _Address.BitList.Bit2;
_DO3.nAddress4 := _Address.BitList.Bit3;
_DO3.nAddress5 := _Address.BitList.Bit4;
_DO3.nAddress6 := _Address.BitList.Bit5;
_DO3.nAddress7 := _Address.BitList.Bit6;

_DO3.bGet := FALSE; // Place action

_DO3.bExecute := TRUE;
IF ConveyorSlideSelect = E_FeedInEmptyBox_PlaceArea.DiffSizeConveyor THEN
	_DO3.bContinue := DiffSizeSlideClear;
ELSIF ConveyorSlideSelect = E_FeedInEmptyBox_PlaceArea.SameSizeConveyor THEN
	_DO3.bContinue := SameSizeSlideClear;
END_IF
M_StartMoveBoxToFeedInConveyor_ClampA := TRUE ; // Method end
END_METHOD

METHOD M_StartMoveBoxToFeedInConveyor_ClampB : BOOL
VAR_INPUT
	ConveyorSlideSelect : E_FeedInEmptyBox_PlaceArea;
    DiffSizeSlideClear  : BOOL;
    SameSizeSlideClear  : BOOL;
END_VAR
VAR_INST
	_Area : ST_IntToBool;
	_Address_ClampB :ST_IntToBool;
END_VAR
// Set target area is round belt
_Area.nInt := E_RobotArea.TransmitCV;
IF ConveyorSlideSelect = E_FeedInEmptyBox_PlaceArea.DiffSizeConveyor THEN
	_Address_ClampB.nInt := 1;
ELSIF ConveyorSlideSelect = E_FeedInEmptyBox_PlaceArea.SameSizeConveyor THEN
	_Address_ClampB.nInt := 2;
ELSE
	// Wrong command, return
	RETURN ;
END_IF
// Send robot target area data
_DO4.nArea1 := _Area.BitList.Bit0;
_DO4.nArea2 := _Area.BitList.Bit1;
_DO4.nArea3 := _Area.BitList.Bit2;
_DO4.nArea4 := _Area.BitList.Bit3;

// Send robot target address data
_DO4.nAddress1 := _Address_ClampB.BitList.Bit0;
_DO4.nAddress2 := _Address_ClampB.BitList.Bit1;
_DO4.nAddress3 := _Address_ClampB.BitList.Bit2;
_DO4.nAddress4 := _Address_ClampB.BitList.Bit3;
_DO4.nAddress5 := _Address_ClampB.BitList.Bit4;
_DO4.nAddress6 := _Address_ClampB.BitList.Bit5;
_DO4.nAddress7 := _Address_ClampB.BitList.Bit6;

_DO4.bGet := FALSE; // Place action

_DO4.bExecute := TRUE;
IF ConveyorSlideSelect = E_FeedInEmptyBox_PlaceArea.DiffSizeConveyor THEN
	_DO4.bContinue := DiffSizeSlideClear;
ELSIF ConveyorSlideSelect = E_FeedInEmptyBox_PlaceArea.SameSizeConveyor THEN
	_DO4.bContinue := SameSizeSlideClear;
END_IF
M_StartMoveBoxToFeedInConveyor_ClampB := TRUE; // Method end
END_METHOD

METHOD M_StartMoveBoxToFeedInConveyor_ClampBoth : BOOL
VAR_INPUT
//    ConveyorSlideSelect : E_FeedInEmptyBox_PlaceArea;
    ClampA_Address      : E_FeedInEmptyBox_PlaceArea;
    ClampB_Address      : E_FeedInEmptyBox_PlaceArea;
	SlideClear_1st : BOOL;
	SlideClear_2nd : BOOL;
END_VAR
VAR_INST
    _Area           : ST_IntToBool;
    _Address_ClampA : ST_IntToBool;
    _Address_ClampB : ST_IntToBool;
END_VAR
// Set target area is round belt
_Area.nInt := E_RobotArea.TransmitCV;
// Select ClampA target address
IF ClampA_Address = E_FeedInEmptyBox_PlaceArea.DiffSizeConveyor THEN
	_Address_ClampA.nInt := 1;
ELSIF ClampA_Address = E_FeedInEmptyBox_PlaceArea.SameSizeConveyor THEN
	_Address_ClampA.nInt := 2;
ELSE
	// Wrong command, return
	RETURN ;
END_IF

// Select ClampB target address
IF ClampB_Address = E_FeedInEmptyBox_PlaceArea.DiffSizeConveyor THEN
	_Address_ClampB.nInt := 1;
ELSIF ClampB_Address = E_FeedInEmptyBox_PlaceArea.SameSizeConveyor THEN
	_Address_ClampB.nInt := 2;
ELSE
	// Wrong command, return
	RETURN;
END_IF

// Send robot target area data
_DO3.nArea1 := _Area.BitList.Bit0;
_DO3.nArea2 := _Area.BitList.Bit1;
_DO3.nArea3 := _Area.BitList.Bit2;
_DO3.nArea4 := _Area.BitList.Bit3;

_DO4.nArea1 := _Area.BitList.Bit0;
_DO4.nArea2 := _Area.BitList.Bit1;
_DO4.nArea3 := _Area.BitList.Bit2;
_DO4.nArea4 := _Area.BitList.Bit3;

// Send robot clampA target address data
_DO3.nAddress1 := _Address_ClampA.BitList.Bit0;
_DO3.nAddress2 := _Address_ClampA.BitList.Bit1;
_DO3.nAddress3 := _Address_ClampA.BitList.Bit2;
_DO3.nAddress4 := _Address_ClampA.BitList.Bit3;
_DO3.nAddress5 := _Address_ClampA.BitList.Bit4;
_DO3.nAddress6 := _Address_ClampA.BitList.Bit5;
_DO3.nAddress7 := _Address_ClampA.BitList.Bit6;

_do4.nAddress1 := _Address_ClampB.BitList.Bit0;
_do4.nAddress2 := _Address_ClampB.BitList.Bit1;
_do4.nAddress3 := _Address_ClampB.BitList.Bit2;
_do4.nAddress4 := _Address_ClampB.BitList.Bit3;
_do4.nAddress5 := _Address_ClampB.BitList.Bit4;
_do4.nAddress6 := _Address_ClampB.BitList.Bit5;
_do4.nAddress7 := _Address_ClampB.BitList.Bit6;


_DO3.bGet := FALSE;
_DO4.bGet := FALSE;

_DO3.bExecute := TRUE;
_DO4.bExecute := TRUE;

_DO3.bContinue := SlideClear_1st;
_DO4.bContinue := SlideClear_2nd;

M_StartMoveBoxToFeedInConveyor_ClampBoth := TRUE; // Method end
END_METHOD

METHOD M_StartMoveBoxToRoundBelt_Both : BOOL
VAR_INPUT
	CarrierSelect_ClampA : E_ReloadRoundBelt_PlaceAddress;
	CarrierSelect_ClampB : E_ReloadRoundBelt_PlaceAddress;
	A2_Sensor : BOOL;
	A3_Sensor : BOOL;
	RoundBeltSafe_1st : BOOL;
	RoundBeltSafe_2nd : BOOL;
END_VAR
VAR_INST
	_Area1 : ST_IntToBool;
	_Address1 : ST_IntToBool;
	CarrierAddress1 :E_ReloadRoundBelt_PlaceAddress;
	_Area2: ST_IntToBool;
	_Address2 : ST_IntToBool;
	CarrierAddress2 :E_ReloadRoundBelt_PlaceAddress;
END_VAR
// Set target area is round belt
_Area1.nInt := E_RobotArea.RoundBelt;
_Area2.nInt := E_RobotArea.RoundBelt;

IF CarrierSelect_ClampA = E_ReloadRoundBelt_PlaceAddress.A2 THEN
	_Address1.nInt := 1;
ELSIF CarrierSelect_ClampA = E_ReloadRoundBelt_PlaceAddress.A3 THEN
	_Address1.nInt := 2;
ELSE
	// Wrong command, return
	RETURN;
END_IF

IF CarrierSelect_ClampB = E_ReloadRoundBelt_PlaceAddress.A2 THEN
	_Address2.nInt := 1;
ELSIF CarrierSelect_ClampB = E_ReloadRoundBelt_PlaceAddress.A3 THEN
	_Address2.nInt := 2;
ELSE
	// Wrong command return
	RETURN;
END_IF
// Send robot target area data
_DO3.nArea1 := _Area1.BitList.Bit0;
_DO3.nArea2 := _Area1.BitList.Bit1;
_DO3.nArea3 := _Area1.BitList.Bit2;
_DO3.nArea4 := _Area1.BitList.Bit3;

_DO4.nArea1 := _Area2.BitList.Bit0;
_DO4.nArea2 := _Area2.BitList.Bit1;
_DO4.nArea3 := _Area2.BitList.Bit2;
_DO4.nArea4 := _Area2.BitList.Bit3;

// Send robot target address data
_DO3.nAddress1 := _Address1.BitList.Bit0;
_DO3.nAddress2 := _Address1.BitList.Bit1;
_DO3.nAddress3 := _Address1.BitList.Bit2;
_DO3.nAddress4 := _Address1.BitList.Bit3;
_DO3.nAddress5 := _Address1.BitList.Bit4;
_DO3.nAddress6 := _Address1.BitList.Bit5;
_DO3.nAddress7 := _Address1.BitList.Bit6;

_DO4.nAddress1 := _Address2.BitList.Bit0;
_DO4.nAddress2 := _Address2.BitList.Bit1;
_DO4.nAddress3 := _Address2.BitList.Bit2;
_DO4.nAddress4 := _Address2.BitList.Bit3;
_DO4.nAddress5 := _Address2.BitList.Bit4;
_DO4.nAddress6 := _Address2.BitList.Bit5;
_DO4.nAddress7 := _Address2.BitList.Bit6;

_DO3.bGet := FALSE; // ClampA Place action
_DO4.bGet := FALSE; // ClampB Place action

IF CarrierSelect_ClampA = E_ReloadRoundBelt_PlaceAddress.A2 THEN
	_DO3.bContinue := NOT A2_Sensor AND RoundBeltSafe_1st;
ELSIF 	CarrierSelect_ClampA = E_ReloadRoundBelt_PlaceAddress.A3 THEN
	_DO3.bContinue := NOT A3_Sensor AND RoundBeltSafe_1st;
END_IF

IF CarrierSelect_ClampB = E_ReloadRoundBelt_PlaceAddress.A2 THEN
	_DO4.bContinue := NOT A2_Sensor AND RoundBeltSafe_2nd;
ELSIF CarrierSelect_ClampB = E_ReloadRoundBelt_PlaceAddress.A3 THEN
	_DO4.bContinue := NOT A3_Sensor AND RoundBeltSafe_2nd;
END_IF

_DO3.bExecute := TRUE; // ClampA Place action
_DO4.bExecute := TRUE; // ClampB Place action


M_StartMoveBoxToRoundBelt_Both := TRUE; // Method end
END_METHOD

METHOD M_StartMoveBoxToRoundBelt_ClampA : BOOL
VAR_INPUT
    CarrierSelect : E_ReloadRoundBelt_PlaceAddress;
    A2_Sensor     : BOOL;
    A3_Sensor     : BOOL;
	RoundBeltSafe : BOOL;
END_VAR
VAR_INST
    _Area          : ST_IntToBool;
    _Address       : ST_IntToBool;
    CarrierAddress : E_ReloadRoundBelt_PlaceAddress;
END_VAR
// Set target area is round belt
_Area.nInt := E_RobotArea.RoundBelt;

IF CarrierSelect = E_ReloadRoundBelt_PlaceAddress.A2 THEN
    _Address.nInt := 1;
ELSIF CarrierSelect = E_ReloadRoundBelt_PlaceAddress.A3 THEN
    _Address.nInt := 2;
ELSE
    // Wrong command, return
    RETURN;
END_IF

// Send robot target area data
_DO3.nArea1 := _Area.BitList.Bit0;
_DO3.nArea2 := _Area.BitList.Bit1;
_DO3.nArea3 := _Area.BitList.Bit2;
_DO3.nArea4 := _Area.BitList.Bit3;

// Send robot target address data
_DO3.nAddress1 := _Address.BitList.Bit0;
_DO3.nAddress2 := _Address.BitList.Bit1;
_DO3.nAddress3 := _Address.BitList.Bit2;
_DO3.nAddress4 := _Address.BitList.Bit3;
_DO3.nAddress5 := _Address.BitList.Bit4;
_DO3.nAddress6 := _Address.BitList.Bit5;
_DO3.nAddress7 := _Address.BitList.Bit6;

_DO3.bGet := FALSE; // Place action

_DO3.bExecute := TRUE;

IF CarrierSelect = E_ReloadRoundBelt_PlaceAddress.A2 THEN
    _DO3.bContinue := NOT A2_Sensor AND RoundBeltSafe ; // Carrier A2 did not has box
ELSIF CarrierSelect = E_ReloadRoundBelt_PlaceAddress.A3 THEN
    _DO3.bContinue := NOT A3_Sensor AND RoundBeltSafe; // Carrier A3 did not has box
END_IF

M_StartMoveBoxToRoundBelt_ClampA := true; // Method end
END_METHOD

METHOD M_StartMoveBoxToRoundBelt_ClampB : BOOL
VAR_INPUT
    CarrierSelect : E_ReloadRoundBelt_PlaceAddress;
    A2_Sensor     : BOOL;
    A3_Sensor     : BOOL;
	RoundBeltSafe : BOOL;
END_VAR
VAR_INST
    _Area          : ST_IntToBool;
    _Address       : ST_IntToBool;
    CarrierAddress : E_ReloadRoundBelt_PlaceAddress;
END_VAR
// Set target area is round belt
_Area.nInt := E_RobotArea.RoundBelt;
IF CarrierSelect = E_ReloadRoundBelt_PlaceAddress.A2 THEN
	_Address.nInt := 1;
ELSIF  CarrierSelect = E_ReloadRoundBelt_PlaceAddress.A3 THEN
	_Address.nInt := 2;
ELSE
	// Wrong command, return
	RETURN ;
END_IF

// Send robot target area data
_DO4.nArea1 := _Area.BitList.Bit0;
_DO4.nArea2 := _Area.BitList.Bit1;
_DO4.nArea3 := _Area.BitList.Bit2;
_DO4.nArea4 := _Area.BitList.Bit3;

// Send robot target address data
_DO4.nAddress1 := _Address.BitList.Bit0;
_DO4.nAddress2 := _Address.BitList.Bit1;
_DO4.nAddress3 := _Address.BitList.Bit2;
_DO4.nAddress4 := _Address.BitList.Bit3;
_DO4.nAddress5 := _Address.BitList.Bit4;
_DO4.nAddress6 := _Address.BitList.Bit5;
_DO4.nAddress7 := _Address.BitList.Bit6;

_DO4.bGet := FALSE; // Place action

_DO4.bExecute := TRUE;

IF CarrierSelect = E_ReloadRoundBelt_PlaceAddress.A2 THEN
	_DO4.bContinue := NOT A2_Sensor AND RoundBeltSafe; // Carrier A2 did not has box
ELSIF CarrierSelect = E_ReloadRoundBelt_PlaceAddress.A3 THEN
	_DO4.bContinue := NOT A3_Sensor AND RoundBeltSafe; // Carrier A3 did not has box
END_IF

M_StartMoveBoxToRoundBelt_ClampB := TRUE; // Method end
END_METHOD

(* This method is used to setting the Fanuc Robot Action " Pickup box from PulloutConveyor , only clampA"
*)
METHOD M_StartPullOutConveyorPickUpBox_ClampA : BOOL
VAR_INPUT
	ClampA_Address : E_PullOutConveyorPosition;
	BoxReady : BOOL; // True : Pullout conveyor box is ready. accroding ClampA target slide is ready or not.
END_VAR
VAR_INST
	_Area : ST_IntToBool;
    _Address_ClampA : ST_IntToBool;
END_VAR
// Set target area is round belt
_Area.nInt := E_RobotArea.PullOutConveyor;
// Select pullout conveyor slide
IF ClampA_Address = E_PullOutConveyorPosition.I3_Slide THEN
	_Address_ClampA.nInt := 1;
ELSIF ClampA_Address = E_PullOutConveyorPosition.I4_Slide THEN
	_Address_ClampA.nInt := 2;
ELSE
	// Wrong command, return
	RETURN ;
END_IF
// Send robot target area data
_DO3.nArea1 := _Area.BitList.Bit0;
_DO3.nArea2 := _Area.BitList.Bit1;
_DO3.nArea3 := _Area.BitList.Bit2;
_DO3.nArea4 := _Area.BitList.Bit3;

// Send robot target address data
_DO3.nAddress1 := _Address_ClampA.BitList.Bit0;
_DO3.nAddress2 := _Address_ClampA.BitList.Bit1;
_DO3.nAddress3 := _Address_ClampA.BitList.Bit2;
_DO3.nAddress4 := _Address_ClampA.BitList.Bit3;
_DO3.nAddress5 := _Address_ClampA.BitList.Bit4;
_DO3.nAddress6 := _Address_ClampA.BitList.Bit5;
_DO3.nAddress7 := _Address_ClampA.BitList.Bit6;

_DO3.bGet := TRUE; // Pickup action
_DO3.bExecute := TRUE;

_DO3.bContinue := BoxReady;

M_StartPullOutConveyorPickUpBox_ClampA := true; // Method end
END_METHOD

(* This method is used to setting the Fanuc Robot Action " Pickup box from PulloutConveyor , only clampB"
*)
METHOD M_StartPullOutConveyorPickUpBox_ClampB : BOOL
VAR_INPUT
	ClampB_Address :E_PullOutConveyorPosition;
	BoxReady : BOOL; // True : Pullout conveyor box is ready. accroding ClampA target slide is ready or not.
END_VAR
VAR_INST
	_Area : ST_IntToBool;
    _Address_ClampB : ST_IntToBool;
END_VAR
// Set target area is round belt
_Area.nInt := E_RobotArea.PullOutConveyor;
// Select pullout conveyor slide
IF ClampB_Address = E_PullOutConveyorPosition.I3_Slide THEN
	_Address_ClampB.nInt := 1;
ELSIF ClampB_Address = E_PullOutConveyorPosition.I4_Slide THEN
	_Address_ClampB.nInt := 2;
ELSE
	// Wrong command, return
	RETURN ;
END_IF

// Send robot target area data
_DO4.nArea1 := _Area.BitList.Bit0;
_DO4.nArea2 := _Area.BitList.Bit1;
_DO4.nArea3 := _Area.BitList.Bit2;
_DO4.nArea4 := _Area.BitList.Bit3;

// Send robot target address data
_DO4.nAddress1 := _Address_ClampB.BitList.Bit0;
_DO4.nAddress2 := _Address_ClampB.BitList.Bit1;
_DO4.nAddress3 := _Address_ClampB.BitList.Bit2;
_DO4.nAddress4 := _Address_ClampB.BitList.Bit3;
_DO4.nAddress5 := _Address_ClampB.BitList.Bit4;
_DO4.nAddress6 := _Address_ClampB.BitList.Bit5;
_DO4.nAddress7 := _Address_ClampB.BitList.Bit6;

_DO4.bGet := TRUE; // Pickup action
_DO4.bExecute := TRUE;

_DO4.bContinue := BoxReady;

M_StartPullOutConveyorPickUpBox_ClampB := true; // Method end
END_METHOD

(* This method is used to setting the Fanuc Robot Action " Pickup box from PulloutConveyor, both clamp"
*)
METHOD M_StartPullOutConveyorPickUpBox_ClampBoth : BOOL
VAR_INPUT
	ClampA_Address : E_PullOutConveyorPosition;
	ClampB_Address : E_PullOutConveyorPosition;
	BoxReady_1 : BOOL; // TRUE : 1st target slide box is ready
	BoxReady_2 : BOOL; // True : 2nd target slide box is ready
END_VAR
VAR_INST
	_Area : ST_IntToBool;
    _Address_ClampA : ST_IntToBool;
    _Address_ClampB : ST_IntToBool;
END_VAR
// Set target area is round belt
_Area.nInt := E_RobotArea.PullOutConveyor;

// Select ClampA target address
IF ClampA_Address = E_PullOutConveyorPosition.I3_Slide THEN
    _Address_ClampA.nInt := 1;
ELSIF ClampA_Address = E_PullOutConveyorPosition.I4_Slide THEN
    _Address_ClampA.nInt := 2;
ELSE
    // Wrong command, return
    RETURN;
END_IF

// Select ClampB target address
IF ClampB_Address = E_PullOutConveyorPosition.I3_Slide THEN
    _Address_ClampB.nInt := 1;
ELSIF ClampB_Address = E_PullOutConveyorPosition.I4_Slide THEN
    _Address_ClampB.nInt := 2;
ELSE
    // Wrong command, return
    RETURN;
END_IF

// Send robot target area data
_DO3.nArea1 := _Area.BitList.Bit0;
_DO3.nArea2 := _Area.BitList.Bit1;
_DO3.nArea3 := _Area.BitList.Bit2;
_DO3.nArea4 := _Area.BitList.Bit3;

_DO4.nArea1 := _Area.BitList.Bit0;
_DO4.nArea2 := _Area.BitList.Bit1;
_DO4.nArea3 := _Area.BitList.Bit2;
_DO4.nArea4 := _Area.BitList.Bit3;

// Send robot target address data
_DO3.nAddress1 := _Address_ClampA.BitList.Bit0;
_DO3.nAddress2 := _Address_ClampA.BitList.Bit1;
_DO3.nAddress3 := _Address_ClampA.BitList.Bit2;
_DO3.nAddress4 := _Address_ClampA.BitList.Bit3;
_DO3.nAddress5 := _Address_ClampA.BitList.Bit4;
_DO3.nAddress6 := _Address_ClampA.BitList.Bit5;
_DO3.nAddress7 := _Address_ClampA.BitList.Bit6;

_DO4.nAddress1 := _Address_ClampB.BitList.Bit0;
_DO4.nAddress2 := _Address_ClampB.BitList.Bit1;
_DO4.nAddress3 := _Address_ClampB.BitList.Bit2;
_DO4.nAddress4 := _Address_ClampB.BitList.Bit3;
_DO4.nAddress5 := _Address_ClampB.BitList.Bit4;
_DO4.nAddress6 := _Address_ClampB.BitList.Bit5;
_DO4.nAddress7 := _Address_ClampB.BitList.Bit6;

_DO3.bGet := TRUE;
_DO4.bGet := TRUE;

_DO3.bExecute := TRUE;
_DO4.bExecute := TRUE;

_DO3.bContinue := BoxReady_1;
_DO4.bContinue := BoxReady_2;

M_StartPullOutConveyorPickUpBox_ClampBoth := true; // Method end
END_METHOD

METHOD PUBLIC M_StartRobotAbsMove : BOOL
VAR_INPUT
	GetBox		: BOOL;
	UseClampA	: BOOL;
	UseClampB   : BOOL;
	Area : E_RobotArea;
	
	
	ClampA_Address	: INT;
	ClampB_Address	: INT;

	BoxReady_1 : BOOL;
	BoxReady_2 : BOOL;
	
END_VAR

VAR_INST
	_Area	: ST_IntToBool;
	_Address_ClampA : ST_IntToBool;
    _Address_ClampB : ST_IntToBool;
END_VAR
//Set target area
_Area.nInt :=Area;

IF UseClampA THEN
	_Address_ClampA.nInt:=ClampA_Address;
	_DO3.nArea1 := _Area.BitList.Bit0;
	_DO3.nArea2 := _Area.BitList.Bit1;
	_DO3.nArea3 := _Area.BitList.Bit2;
	_DO3.nArea4 := _Area.BitList.Bit3;

	_DO3.nAddress1 := _Address_ClampA.BitList.Bit0;
	_DO3.nAddress2 := _Address_ClampA.BitList.Bit1;
	_DO3.nAddress3 := _Address_ClampA.BitList.Bit2;
	_DO3.nAddress4 := _Address_ClampA.BitList.Bit3;
	_DO3.nAddress5 := _Address_ClampA.BitList.Bit4;
	_DO3.nAddress6 := _Address_ClampA.BitList.Bit5;
	_DO3.nAddress7 := _Address_ClampA.BitList.Bit6;
	_DO3.bGet := GetBox;
	_DO3.bExecute := TRUE;
	_DO3.bContinue := BoxReady_1;	
END_IF

IF UseClampB THEN
	_Address_ClampB.nInt:=ClampB_Address;
	_DO4.nArea1 := _Area.BitList.Bit0;
	_DO4.nArea2 := _Area.BitList.Bit1;
	_DO4.nArea3 := _Area.BitList.Bit2;
	_DO4.nArea4 := _Area.BitList.Bit3;
	
	_DO4.nAddress1 := _Address_ClampB.BitList.Bit0;
	_DO4.nAddress2 := _Address_ClampB.BitList.Bit1;
	_DO4.nAddress3 := _Address_ClampB.BitList.Bit2;
	_DO4.nAddress4 := _Address_ClampB.BitList.Bit3;
	_DO4.nAddress5 := _Address_ClampB.BitList.Bit4;
	_DO4.nAddress6 := _Address_ClampB.BitList.Bit5;
	_DO4.nAddress7 := _Address_ClampB.BitList.Bit6;
	_DO4.bGet := GetBox;
	_DO4.bExecute := TRUE;
	_DO4.bContinue := BoxReady_2;	
END_IF

M_StartRobotAbsMove :=TRUE;




















M_StartRobotAbsMove:=TRUE;
END_METHOD

METHOD M_StartWarehouseMoveAction_ClampA : BOOL
VAR_INPUT
	WareHouseSelect : E_WareHouse;
	Info : ST_WareHouseCoordinates; // Input Warehouse with robot move parameter for pickup box;
	ClampAction :E_ClampAction;
	BoxReady : BOOL;
END_VAR
VAR_OUTPUT
	Error : BOOL;
	ErrMsg :T_MaxString;
END_VAR
VAR_INST
	_Layer : ST_IntToBool;
	_Slide : ST_IntToBool;
END_VAR
// Set target warehouse
CASE WareHouseSelect OF
    E_WareHouse.WareHouseA:
        _DO1.bTargetWareHouseA := TRUE;
        _DO1.bTargetWareHouseB := FALSE;
    E_WareHouse.WareHouseB:
        _DO1.bTargetWareHouseA := FALSE;
        _DO1.bTargetWareHouseB := TRUE;
ELSE
    _DO1.bTargetWareHouseA := FALSE;
    _DO1.bTargetWareHouseB := FALSE;
    Error                  := TRUE;
    ErrMsg                 := 'ClampA target warehouse out of range';
	RETURN;
END_CASE

// Set Warehouse coordinates
_Layer.nInt := info.Layer;
_Slide.nInt := info.Slide;

// Send Layer data to robot
_DO1.nLayer1 := _Layer.BitList.Bit0;
_DO1.nLayer2 := _Layer.BitList.Bit1;
_DO1.nLayer3 := _Layer.BitList.Bit2;
_DO1.nLayer4 := _Layer.BitList.Bit3;

// Send Slide data to Robot
_DO1.nSlide1 := _Slide.BitList.Bit0;
_DO1.nSlide2 := _Slide.BitList.Bit1;
_DO1.nSlide3 := _Slide.BitList.Bit2;
_DO1.nSlide4 := _Slide.BitList.Bit3;
_DO1.nSlide5 := _Slide.BitList.Bit4;

// Send clamp action to robot
CASE ClampAction OF
	E_ClampAction.PickUp:
		_DO1.bGet := TRUE;
	E_ClampAction.Place:
		_DO1.bGet := FALSE;
ELSE
	Error := TRUE;
	ErrMsg := 'Clamp action not defined';
	RETURN;
END_CASE

// Send action data to robot
_DO1.bExecute := NOT Error;
_DO1.bContinue := BoxReady;
M_StartWarehouseMoveAction_ClampA := NOT Error; // Method end
END_METHOD

METHOD M_StartWarehouseMoveAction_ClampB : BOOL
VAR_INPUT
	WareHouseSelect : E_WareHouse;
	Info : ST_WareHouseCoordinates; // Input Warehouse with robot move parameter for pickup box;
	ClampAction :E_ClampAction;
	BoxReady : BOOL;
END_VAR
VAR_OUTPUT
	Error : BOOL;
	ErrMsg :T_MaxString;
END_VAR
VAR_INST
	_Layer : ST_IntToBool;
	_Slide : ST_IntToBool;
END_VAR
// Set target warehouse
CASE WareHouseSelect OF
    E_WareHouse.WareHouseA:
        _DO2.bTargetWareHouseA := TRUE;
        _DO2.bTargetWareHouseB := FALSE;
    E_WareHouse.WareHouseB:
        _DO2.bTargetWareHouseA := FALSE;
        _DO2.bTargetWareHouseB := TRUE;
ELSE
    _DO2.bTargetWareHouseA := FALSE;
    _DO2.bTargetWareHouseB := FALSE;
    Error                  := TRUE;
    ErrMsg                 := 'ClampB target warehouse out of range';
	RETURN;
END_CASE

// Set Warehouse coordinates
_Layer.nInt := info.Layer;
_Slide.nInt := info.Slide;

// Send Layer data to robot
_DO2.nLayer1 := _Layer.BitList.Bit0;
_DO2.nLayer2 := _Layer.BitList.Bit1;
_DO2.nLayer3 := _Layer.BitList.Bit2;
_DO2.nLayer4 := _Layer.BitList.Bit3;

// Send Slide data to Robot
_DO2.nSlide1 := _Slide.BitList.Bit0;
_DO2.nSlide2 := _Slide.BitList.Bit1;
_DO2.nSlide3 := _Slide.BitList.Bit2;
_DO2.nSlide4 := _Slide.BitList.Bit3;
_DO2.nSlide5 := _Slide.BitList.Bit4;

// Send clamp action to robot
CASE ClampAction OF
	E_ClampAction.PickUp:
		_DO2.bGet := TRUE;
	E_ClampAction.Place:
		_DO2.bGet := FALSE;
ELSE
	Error := TRUE;
	ErrMsg := 'Clamp action not defined';
	RETURN;
END_CASE

// Send action data to robot
_DO2.bExecute := NOT Error;
_DO2.bContinue := BoxReady;

M_StartWarehouseMoveAction_ClampB := NOT Error; // Method End
END_METHOD

METHOD M_StartWarehouseMoveAction_ClampBoth : BOOL
VAR_INPUT
	WareHouseSelect : E_WareHouse;
	ClampA_Info : ST_WareHouseCoordinates; // Input Warehouse with robot move parameter for pickup box;
	ClampB_Info : ST_WareHouseCoordinates; // Input Warehouse with robot move parameter for pickup box;
	ClampAction_A : E_ClampAction;
	ClampAction_B : E_ClampAction;
	BoxReady_1st : BOOL; // Box is arrived, ready to pickup
	BoxReady_2nd : BOOL; // Box is arrived, ready to pickup
END_VAR
VAR_OUTPUT
	Error : BOOL;
	ErrMsg :T_MaxString;
END_VAR
VAR_INST
	_LayerClampA :ST_IntToBool;
	_SlideClampA : ST_IntToBool;
	_LayerClampB : ST_IntToBool;
	_SLideClampB : ST_IntToBool;
END_VAR
// Set target warehouse
CASE WareHouseSelect OF
    E_WareHouse.WareHouseA:
        _DO1.bTargetWareHouseA := TRUE;
        _DO1.bTargetWareHouseB := FALSE;
        _DO2.bTargetWareHouseA := TRUE;
        _DO2.bTargetWareHouseB := FALSE;
    E_WareHouse.WareHouseB:
        _DO1.bTargetWareHouseA := FALSE;
        _DO1.bTargetWareHouseB := TRUE;
        _DO2.bTargetWareHouseA := FALSE;
        _DO2.bTargetWareHouseB := TRUE;
ELSE
    _DO1.bTargetWareHouseA := FALSE;
    _DO1.bTargetWareHouseB := FALSE;
    _DO2.bTargetWareHouseA := FALSE;
    _DO2.bTargetWareHouseB := FALSE;
    Error                  := TRUE;
    ErrMsg                 := 'Clamp target warehouse out of range';
    RETURN;
END_CASE

// Assign coordinates 
_LayerClampA.nInt := ClampA_Info.Layer;
_SlideClampA.nInt := ClampA_Info.Slide;
_LayerClampB.nInt := ClampB_Info.Layer;
_SlideClampB.nInt := ClampB_Info.Slide;

// Send Layer data to Robot
_DO1.nLayer1 := _LayerClampA.BitList.Bit0;
_DO1.nLayer2 := _LayerClampA.BitList.Bit1;
_DO1.nLayer3 := _LayerClampA.BitList.Bit2;
_DO1.nLayer4 := _LayerClampA.BitList.Bit3;
_DO2.nLayer1 := _LayerClampB.BitList.Bit0;
_DO2.nLayer2 := _LayerClampB.BitList.Bit1;
_DO2.nLayer3 := _LayerClampB.BitList.Bit2;
_DO2.nLayer4 := _LayerClampB.BitList.Bit3;
// Send Slide data to Robot
_DO1.nSlide1 := _SlideClampA.BitList.Bit0;
_DO1.nSlide2 := _SlideClampA.BitList.Bit1;
_DO1.nSlide3 := _SlideClampA.BitList.Bit2;
_DO1.nSlide4 := _SlideClampA.BitList.Bit3;
_DO1.nSlide5 := _SlideClampA.BitList.Bit4;

_DO2.nSlide1 := _SlideClampB.BitList.Bit0;
_DO2.nSlide2 := _SlideClampB.BitList.Bit1;
_DO2.nSlide3 := _SlideClampB.BitList.Bit2;
_DO2.nSlide4 := _SlideClampB.BitList.Bit3;
_DO2.nSlide5 := _SlideClampB.BitList.Bit4;

// Set clamp action 
CASE ClampAction_A OF
	E_ClampAction.PickUp:
		_DO1.bGet := TRUE;
	E_ClampAction.Place:
		_DO1.bGet := FALSE;
ELSE
	Error := TRUE;
	ErrMsg := 'ClampA action not defined';
	RETURN;
END_CASE

// Set clamp action
CASE ClampAction_B OF
	E_ClampAction.PickUp:
		_DO2.bGet := TRUE;
	E_ClampAction.Place:
		_DO2.bGet := FALSE;
ELSE
	Error := TRUE;
	ErrMsg := 'ClampB action not defined';
	RETURN;	
END_CASE

// set execute
_DO1.bExecute := NOT Error;
_DO2.bExecute := NOT Error;

_DO1.bContinue := BoxReady_1st;
_DO2.bContinue := BoxReady_2nd;

M_StartWarehouseMoveAction_ClampBoth := NOT Error; // Method end
END_METHOD

METHOD M_StartWareHousePickUpBox_ClampA : Bool
VAR_INPUT
	WareHouseSelect : E_WareHouse;
	Info : ST_WareHouseCoordinates; // Input Warehouse with robot move parameter for pickup box;
	BoxReady_1st : BOOL;
END_VAR
VAR_INST
	_Layer : ST_IntToBool;
	_Slide : ST_IntToBool;
END_VAR
// Send target warehouse to robot
IF WareHouseSelect = E_WareHouse.WareHouseA THEN
	_DO1.bTargetWareHouseA := TRUE;
	_DO1.bTargetWareHouseB := FALSE;
ELSIF WareHouseSelect = E_WareHouse.WareHouseB THEN
	_DO1.bTargetWareHouseA := FALSE;
	_DO1.bTargetWareHouseB := TRUE;
ELSE
	_DO1.bTargetWareHouseA := FALSE;
	_DO1.bTargetWareHouseB := FALSE;
END_IF

// Assign coordinates 
_Layer.nInt := info.Layer;
_Slide.nInt := info.Slide;

// Send Layer data to Robot
_DO1.nLayer1 := _Layer.BitList.Bit0;
_DO1.nLayer2 := _Layer.BitList.Bit1;
_DO1.nLayer3 := _Layer.BitList.Bit2;
_DO1.nLayer4 := _Layer.BitList.Bit3;

// Send Slide data to Robot
_DO1.nSlide1 := _Slide.BitList.Bit0;
_DO1.nSlide2 := _Slide.BitList.Bit1;
_DO1.nSlide3 := _Slide.BitList.Bit2;
_DO1.nSlide4 := _Slide.BitList.Bit3;
_DO1.nSlide5 := _Slide.BitList.Bit4;

// Send action data to robot
_DO1.bGet := TRUE; // PickUp
// Send execute command 
_DO1.bExecute := TRUE;
_DO1.bContinue := BoxReady_1st;
M_StartWareHousePickUpBox_ClampA := TRUE; // Method end
END_METHOD

METHOD M_StartWareHousePickUpBox_ClampB : BOOL
VAR_INPUT
	WareHouseSelect : E_WareHouse;
	Info : ST_WareHouseCoordinates; // Input Warehouse with robot move parameter for pickup box;
	BoxReady_2nd : BOOL;
END_VAR
VAR_INST
	_Layer : ST_IntToBool;
	_Slide : ST_IntToBool;
END_VAR
// Send target warehouse to robot
IF WareHouseSelect = E_WareHouse.WareHouseA THEN
    _DO2.bTargetWareHouseA := TRUE;
    _DO2.bTargetWareHouseB := FALSE;
ELSIF WareHouseSelect = E_WareHouse.WareHouseB THEN
    _DO2.bTargetWareHouseA := FALSE;
    _DO2.bTargetWareHouseB := TRUE;
ELSE
    _DO2.bTargetWareHouseA := FALSE;
    _DO2.bTargetWareHouseB := FALSE;
END_IF

// Assign coordinates 
_Layer.nInt := info.Layer;
_Slide.nInt := info.Slide;

// Send Layer data to Robot
_DO2.nLayer1 := _Layer.BitList.Bit0;
_DO2.nLayer2 := _Layer.BitList.Bit1;
_DO2.nLayer3 := _Layer.BitList.Bit2;
_DO2.nLayer4 := _Layer.BitList.Bit3;

// Send Slide data to Robot
_DO2.nSlide1 := _Slide.BitList.Bit0;
_DO2.nSlide2 := _Slide.BitList.Bit1;
_DO2.nSlide3 := _Slide.BitList.Bit2;
_DO2.nSlide4 := _Slide.BitList.Bit3;
_DO2.nSlide5 := _Slide.BitList.Bit4;

// Send action data to robot
_DO2.bGet := TRUE; // PickUp
// Send execute command 
_DO2.bExecute := TRUE;
_DO2.bContinue:=BoxReady_2nd;
M_StartWareHousePickUpBox_ClampB := TRUE; // Method end
END_METHOD

METHOD M_StartWareHousePickUpBox_ClampBoth : BOOL
VAR_INPUT
	WareHouseSelect : E_WareHouse;
	ClampA_Info : ST_WareHouseCoordinates; // Input Warehouse with robot move parameter for pickup box;
	ClampB_Info : ST_WareHouseCoordinates; // Input Warehouse with robot move parameter for pickup box;
	BoxReady_1st : BOOL; // Box is arrived, ready to pickup
	BoxReady_2nd : BOOL; // Box is arrived, ready to pickup
END_VAR
VAR_OUTPUT
	Error : BOOL;
	ErrMsg :T_MaxString;
END_VAR
VAR_INST
	_LayerClampA : ST_IntToBool;
	_SlideClampA : ST_IntToBool;
	_LayerClampB : ST_IntToBool;
	_SlideClampB : ST_IntToBool;
END_VAR
// Set target warehouse
CASE WareHouseSelect OF
    E_WareHouse.WareHouseA:
        _DO1.bTargetWareHouseA := TRUE;
        _DO1.bTargetWareHouseB := FALSE;
        _DO2.bTargetWareHouseA := TRUE;
        _DO2.bTargetWareHouseB := FALSE;
    E_WareHouse.WareHouseB:
        _DO1.bTargetWareHouseA := FALSE;
        _DO1.bTargetWareHouseB := TRUE;
        _DO2.bTargetWareHouseA := FALSE;
        _DO2.bTargetWareHouseB := TRUE;
ELSE
    _DO1.bTargetWareHouseA := FALSE;
    _DO1.bTargetWareHouseB := FALSE;
    _DO2.bTargetWareHouseA := FALSE;
    _DO2.bTargetWareHouseB := FALSE;
    Error                  := TRUE;
    ErrMsg                 := 'Clamp target warehouse out of range';
    RETURN;
END_CASE

// Assign coordinates 
_LayerClampA.nInt := ClampA_Info.Layer;
_SlideClampA.nInt := ClampA_Info.Slide;
_LayerClampB.nInt := ClampB_Info.Layer;
_SlideClampB.nInt := ClampB_Info.Slide;

// Send Layer data to Robot
_DO1.nLayer1 := _LayerClampA.BitList.Bit0;
_DO1.nLayer2 := _LayerClampA.BitList.Bit1;
_DO1.nLayer3 := _LayerClampA.BitList.Bit2;
_DO1.nLayer4 := _LayerClampA.BitList.Bit3;

_DO2.nLayer1 := _LayerClampB.BitList.Bit0;
_DO2.nLayer2 := _LayerClampB.BitList.Bit1;
_DO2.nLayer3 := _LayerClampB.BitList.Bit2;
_DO2.nLayer4 := _LayerClampB.BitList.Bit3;
// Send Slide data to Robot
_DO1.nSlide1 := _SlideClampA.BitList.Bit0;
_DO1.nSlide2 := _SlideClampA.BitList.Bit1;
_DO1.nSlide3 := _SlideClampA.BitList.Bit2;
_DO1.nSlide4 := _SlideClampA.BitList.Bit3;
_DO1.nSlide5 := _SlideClampA.BitList.Bit4;

_DO2.nSlide1 := _SlideClampB.BitList.Bit0;
_DO2.nSlide2 := _SlideClampB.BitList.Bit1;
_DO2.nSlide3 := _SlideClampB.BitList.Bit2;
_DO2.nSlide4 := _SlideClampB.BitList.Bit3;
_DO2.nSlide5 := _SlideClampB.BitList.Bit4;

// Send action data to robot
_DO1.bGet := TRUE; // ClampA PickUp
_DO2.bGet := TRUE; // ClampB PickUp
// Send execute command 
_DO1.bExecute := NOT Error;
_DO2.bExecute := NOT Error;

_DO1.bContinue := BoxReady_1st;
_DO2.bContinue := BoxReady_2nd;

M_StartWareHousePickUpBox_ClampBoth := NOT Error; // Method end
END_METHOD

METHOD M_StartWareHousePlaceBox_ClampA : Bool
VAR_INPUT
	WareHouseSelect : E_WareHouse;
	Info : ST_WareHouseCoordinates; // Input Warehouse with robot move parameter for pickup box;
	BoxReady_1st : BOOL;
END_VAR
VAR_INST
	_Layer : ST_IntToBool;
	_Slide : ST_IntToBool;
END_VAR
// Send target warehouse to robot
IF WareHouseSelect = E_WareHouse.WareHouseA THEN
	_DO1.bTargetWareHouseA := TRUE;
	_DO1.bTargetWareHouseB := FALSE;
ELSIF WareHouseSelect = E_WareHouse.WareHouseB THEN
	_DO1.bTargetWareHouseA := FALSE;
	_DO1.bTargetWareHouseB := TRUE;
ELSE
	_DO1.bTargetWareHouseA := FALSE;
	_DO1.bTargetWareHouseB := FALSE;
END_IF

// Assign coordinates 
_Layer.nInt := info.Layer;
_Slide.nInt := info.Slide;

// Send Layer data to Robot
_DO1.nLayer1 := _Layer.BitList.Bit0;
_DO1.nLayer2 := _Layer.BitList.Bit1;
_DO1.nLayer3 := _Layer.BitList.Bit2;
_DO1.nLayer4 := _Layer.BitList.Bit3;

// Send Slide data to Robot
_DO1.nSlide1 := _Slide.BitList.Bit0;
_DO1.nSlide2 := _Slide.BitList.Bit1;
_DO1.nSlide3 := _Slide.BitList.Bit2;
_DO1.nSlide4 := _Slide.BitList.Bit3;
_DO1.nSlide5 := _Slide.BitList.Bit4;

// Send action data to robot
_DO1.bGet := FALSE; // PickUp
// Send execute command 
_DO1.bExecute := TRUE;
_DO1.bContinue := BoxReady_1st;
M_StartWareHousePlaceBox_ClampA := TRUE; // Method end
END_METHOD

METHOD M_StartWareHousePlaceBox_ClampB : BOOL
VAR_INPUT
	WareHouseSelect : E_WareHouse;
	Info : ST_WareHouseCoordinates; // Input Warehouse with robot move parameter for pickup box;
	BoxReady_2nd : BOOL;
END_VAR
VAR_INST
	_Layer : ST_IntToBool;
	_Slide : ST_IntToBool;
END_VAR
// Send target warehouse to robot
IF WareHouseSelect = E_WareHouse.WareHouseA THEN
    _DO2.bTargetWareHouseA := TRUE;
    _DO2.bTargetWareHouseB := FALSE;
ELSIF WareHouseSelect = E_WareHouse.WareHouseB THEN
    _DO2.bTargetWareHouseA := FALSE;
    _DO2.bTargetWareHouseB := TRUE;
ELSE
    _DO2.bTargetWareHouseA := FALSE;
    _DO2.bTargetWareHouseB := FALSE;
END_IF

// Assign coordinates 
_Layer.nInt := info.Layer;
_Slide.nInt := info.Slide;

// Send Layer data to Robot
_DO2.nLayer1 := _Layer.BitList.Bit0;
_DO2.nLayer2 := _Layer.BitList.Bit1;
_DO2.nLayer3 := _Layer.BitList.Bit2;
_DO2.nLayer4 := _Layer.BitList.Bit3;

// Send Slide data to Robot
_DO2.nSlide1 := _Slide.BitList.Bit0;
_DO2.nSlide2 := _Slide.BitList.Bit1;
_DO2.nSlide3 := _Slide.BitList.Bit2;
_DO2.nSlide4 := _Slide.BitList.Bit3;
_DO2.nSlide5 := _Slide.BitList.Bit4;

// Send action data to robot
_DO2.bGet := FALSE; // PickUp
// Send execute command 
_DO2.bExecute := TRUE;
_DO2.bContinue:=BoxReady_2nd;
M_StartWareHousePlaceBox_ClampB := TRUE; // Method end
END_METHOD

METHOD M_StartWareHousePlaceUpBox_ClampBoth : BOOL
VAR_INPUT
	WareHouseSelect : E_WareHouse;
	ClampA_Info : ST_WareHouseCoordinates; // Input Warehouse with robot move parameter for pickup box;
	ClampB_Info : ST_WareHouseCoordinates; // Input Warehouse with robot move parameter for pickup box;
	BoxReady_1st : BOOL; // Box is arrived, ready to pickup
	BoxReady_2nd : BOOL; // Box is arrived, ready to pickup
END_VAR
VAR_OUTPUT
	Error : BOOL;
	ErrMsg :T_MaxString;
END_VAR
VAR_INST
	_LayerClampA : ST_IntToBool;
	_SlideClampA : ST_IntToBool;
	_LayerClampB : ST_IntToBool;
	_SlideClampB : ST_IntToBool;
END_VAR
// Set target warehouse
CASE WareHouseSelect OF
    E_WareHouse.WareHouseA:
        _DO1.bTargetWareHouseA := TRUE;
        _DO1.bTargetWareHouseB := FALSE;
        _DO2.bTargetWareHouseA := TRUE;
        _DO2.bTargetWareHouseB := FALSE;
    E_WareHouse.WareHouseB:
        _DO1.bTargetWareHouseA := FALSE;
        _DO1.bTargetWareHouseB := TRUE;
        _DO2.bTargetWareHouseA := FALSE;
        _DO2.bTargetWareHouseB := TRUE;
ELSE
    _DO1.bTargetWareHouseA := FALSE;
    _DO1.bTargetWareHouseB := FALSE;
    _DO2.bTargetWareHouseA := FALSE;
    _DO2.bTargetWareHouseB := FALSE;
    Error                  := TRUE;
    ErrMsg                 := 'Clamp target warehouse out of range';
    RETURN;
END_CASE

// Assign coordinates 
_LayerClampA.nInt := ClampA_Info.Layer;
_SlideClampA.nInt := ClampA_Info.Slide;
_LayerClampB.nInt := ClampB_Info.Layer;
_SlideClampB.nInt := ClampB_Info.Slide;

// Send Layer data to Robot
_DO1.nLayer1 := _LayerClampA.BitList.Bit0;
_DO1.nLayer2 := _LayerClampA.BitList.Bit1;
_DO1.nLayer3 := _LayerClampA.BitList.Bit2;
_DO1.nLayer4 := _LayerClampA.BitList.Bit3;

_DO2.nLayer1 := _LayerClampB.BitList.Bit0;
_DO2.nLayer2 := _LayerClampB.BitList.Bit1;
_DO2.nLayer3 := _LayerClampB.BitList.Bit2;
_DO2.nLayer4 := _LayerClampB.BitList.Bit3;
// Send Slide data to Robot
_DO1.nSlide1 := _SlideClampA.BitList.Bit0;
_DO1.nSlide2 := _SlideClampA.BitList.Bit1;
_DO1.nSlide3 := _SlideClampA.BitList.Bit2;
_DO1.nSlide4 := _SlideClampA.BitList.Bit3;
_DO1.nSlide5 := _SlideClampA.BitList.Bit4;

_DO2.nSlide1 := _SlideClampB.BitList.Bit0;
_DO2.nSlide2 := _SlideClampB.BitList.Bit1;
_DO2.nSlide3 := _SlideClampB.BitList.Bit2;
_DO2.nSlide4 := _SlideClampB.BitList.Bit3;
_DO2.nSlide5 := _SlideClampB.BitList.Bit4;

// Send action data to robot
_DO1.bGet := FALSE; // ClampA PickUp
_DO2.bGet := FALSE; // ClampB PickUp
// Send execute command 
_DO1.bExecute := NOT Error;
_DO2.bExecute := NOT Error;

_DO1.bContinue := BoxReady_1st;
_DO2.bContinue := BoxReady_2nd;

M_StartWareHousePlaceUpBox_ClampBoth := NOT Error; // Method end
END_METHOD

METHOD M_SwitchRSR3 : BOOL
VAR_INPUT
END_VAR
END_METHOD

PROPERTY Read_OffsetP : INT
GET
Read_OffsetP := _DI6;
END_GET
END_PROPERTY

PROPERTY Read_OffsetR : INT
GET
Read_OffsetR := _DI7;
END_GET
END_PROPERTY

PROPERTY Read_OffsetW : INT
GET
Read_OffsetW := _DI5;
END_GET
END_PROPERTY

PROPERTY Read_OffsetX : INT
GET
Read_OffsetX := _DI2;
END_GET
END_PROPERTY

PROPERTY Read_OffsetY : INT
GET
Read_OffsetY := _DI3;
END_GET
END_PROPERTY

PROPERTY Read_OffsetZ : INT
GET
Read_OffsetZ := _DI4;
END_GET
END_PROPERTY

PROPERTY ReadDataCommand : BOOL;
SET
_DO6.ReadPara_Execute := BOOL_TO_BIT(ReadDataCommand);
END_SET
END_PROPERTY

PROPERTY ReadWrite_Address : Int
SET
_Do14 := ReadWrite_Address;
END_SET
END_PROPERTY

PROPERTY ReadWrite_Area : E_RobotArea
SET
_Do13 := ReadWrite_Area;
END_SET
END_PROPERTY

(* This variable is used to define read/write offset data clamp A
*)
PROPERTY ReadWrite_ClampA : BOOL
SET
_DO6.ClampA :=  BOOL_TO_BIT(ReadWrite_ClampA );
END_SET
END_PROPERTY

(* This variable is used to define read/write offset data clamp B
*)
PROPERTY ReadWrite_ClampB : BOOL
SET
_DO6.ClampB :=BOOL_TO_BIT( ReadWrite_ClampB);
END_SET
END_PROPERTY

(* This variable is used to define read/write offset data warehouse A
*)
PROPERTY ReadWrite_WareHouseA : BOOL
SET
_DO6.WareHouseA := BOOL_TO_BIT(ReadWrite_WareHouseA);
END_SET
END_PROPERTY

(* This variable is used to define read/write offset data warehouse B
*)
PROPERTY ReadWrite_WareHouseB : BOOL
SET
_DO6.WarehouseB := BOOL_TO_BIT(ReadWrite_WareHouseB);
END_SET
END_PROPERTY

(*Fanuc robot ready to work for command (Warehouse、AbsMove)*)
PROPERTY ReadyOperation : Bool
GET
ReadyOperation := _RSR1_Ready;
END_GET
END_PROPERTY

PROPERTY ReadySetParameter : Bool
GET
ReadySetParameter := _RSR3_Ready;
END_GET
END_PROPERTY

METHOD ReBoot
VAR_INPUT
END_VAR
eState := E_MethodStatus_Basic.STATE_DORMANT;
END_METHOD

PROPERTY SlideIndex : INT
SET
_DO16 := SlideIndex;
END_SET
END_PROPERTY

PROPERTY Status : ST_FanucUI1
GET
Status := _UI1;
END_GET
END_PROPERTY

METHOD Update : BOOL
VAR_INPUT
END_VAR
// Robot -> PLC 4 byte 外圍設備Output(Fanuc Robot的外圍)
MEMMOVE(
destAddr:=ADR(_UO1)
,srcAddr:=ADR(_rawIn_UI[0])
,n:=4
);

// PLC -> Robot 外圍設備Input(Fanuc Robot的外圍)
MEMMOVE(
destAddr:=ADR(_rawOut_UO[0])
,srcAddr:=ADR(_UI1)
,n:=4
);
// PLC -> Robot Digital Output 2byte(send the command to Fanuc Robot), Warehouse Robot move ClampA
MEMMOVE(
destAddr:=ADR(_rawOut_DO[0])
,srcAddr:=ADR(_DO1)
,n:=2 
);
// PLC -> Robot Digital Output 2byte(send the command to Fanuc Robot), Warehouse Robot move ClampB
MEMMOVE(
destAddr:=ADR(_rawOut_DO[2])
,srcAddr:=ADR(_DO2)
,n:=2 
);
// PLC -> Robot Digital Output 2byte(send the command to Fanuc Robot), ABS Robot move ClampA
MEMMOVE(
destAddr:=ADR(_rawOut_DO[4])
,srcAddr:=ADR(_DO3)
,n:=2 
);
// PLC -> Robot Digital Output 2byte(send the command to Fanuc Robot), ABS Robot move ClampA
MEMMOVE(
destAddr:=ADR(_rawOut_DO[6])
,srcAddr:=ADR(_DO4)
,n:=2 
);
// PLC -> Robot Digital output 2byte(send the command to Fanuc Robot), General Command
MEMMOVE(
destAddr:=ADR(_rawOut_DO[8])
,srcAddr:=ADR(_DO5)
,n:=2 
);
MEMMOVE(
destAddr:=ADR(_rawOut_DO[10])
,srcAddr:=ADR(_DO6)
,n:=2 
);
MEMMOVE(
destAddr:=ADR(_rawOut_DO[12])
,srcAddr:=ADR(_DO7)
,n:=2 
);
MEMMOVE(
destAddr:=ADR(_rawOut_DO[14])
,srcAddr:=ADR(_DO8)
,n:=2 
);
MEMMOVE(
destAddr:=ADR(_rawOut_DO[16])
,srcAddr:=ADR(_DO9)
,n:=2 
);

MEMMOVE(
destAddr:=ADR(_rawOut_DO[18])
,srcAddr:=ADR(_DO10)
,n:=2 
);
MEMMOVE(
destAddr:=ADR(_rawOut_DO[20])
,srcAddr:=ADR(_DO11)
,n:=2 
);
MEMMOVE(
destAddr:=ADR(_rawOut_DO[22])
,srcAddr:=ADR(_DO12)
,n:=2 
);
MEMMOVE(
destAddr:=ADR(_rawOut_DO[24])
,srcAddr:=ADR(_DO13)
,n:=2 
);
MEMMOVE(
destAddr:=ADR(_rawOut_DO[26])
,srcAddr:=ADR(_DO14)
,n:=2 
);
MEMMOVE(
destAddr:=ADR(_rawOut_DO[28])
,srcAddr:=ADR(_DO15)
,n:=2 
);
MEMMOVE(
destAddr:=ADR(_rawOut_DO[30])
,srcAddr:=ADR(_DO16)
,n:=2 
);


// Robot -> PLC Digital Input 3byte(Send Robot Status to PLC), All service
MEMMOVE(
destAddr:=ADR(_DI1)
,srcAddr:=ADR(_rawIn_DI[0])
,n:=3
);

MEMMOVE(
destAddr:=ADR(_DI2)
,srcAddr:=ADR(_rawIn_DI[3])
,n:=2
);
MEMMOVE(
destAddr:=ADR(_DI3)
,srcAddr:=ADR(_rawIn_DI[5])
,n:=2
);
MEMMOVE(
destAddr:=ADR(_DI4)
,srcAddr:=ADR(_rawIn_DI[7])
,n:=2
);
MEMMOVE(
destAddr:=ADR(_DI5)
,srcAddr:=ADR(_rawIn_DI[9])
,n:=2
);
MEMMOVE(
destAddr:=ADR(_DI6)
,srcAddr:=ADR(_rawIn_DI[11])
,n:=2
);
MEMMOVE(
destAddr:=ADR(_DI7)
,srcAddr:=ADR(_rawIn_DI[13])
,n:=2
);
MEMMOVE(
destAddr:=ADR(_DI8)
,srcAddr:=ADR(_rawIn_DI[15])
,n:=2
);
MEMMOVE(
destAddr:=ADR(_DI9)
,srcAddr:=ADR(_rawIn_DI[17])
,n:=2
);
MEMMOVE(
destAddr:=ADR(_DI10)
,srcAddr:=ADR(_rawIn_DI[19])
,n:=2
);
MEMMOVE(
destAddr:=ADR(_DI11)
,srcAddr:=ADR(_rawIn_DI[21])
,n:=2
);
MEMMOVE(
destAddr:=ADR(_DI12)
,srcAddr:=ADR(_rawIn_DI[23])
,n:=2
);

// Robot Status com
qEnable:=_UO1.UO01_CmdEnabled AND _UO1.UO02_SystemReady;
Error:=Fault();

// Velocity Command transfer
_DO5.VelocityBit0 := _VelocityCommand.BitList.Bit0;
_DO5.VelocityBit1 := _VelocityCommand.BitList.Bit1;
_DO5.VelocityBit2 := _VelocityCommand.BitList.Bit2;
_DO5.VelocityBit3 := _VelocityCommand.BitList.Bit3;
_DO5.VelocityBit4 := _VelocityCommand.BitList.Bit4;
_DO5.VelocityBit5 := _VelocityCommand.BitList.Bit5;
_DO5.VelocityBit6 := _VelocityCommand.BitList.Bit6;
_DO5.VelocityBit7 := _VelocityCommand.BitList.Bit7;
END_METHOD

{attribute 'monitoring' := 'variable'}
PROPERTY VelocityCommand : Int
GET
VelocityCommand :=_VelocityCommand.nInt;
END_GET
SET
_VelocityCommand.nInt :=VelocityCommand;
END_SET
END_PROPERTY

PROPERTY WareHouseClampA_Handshake : ST_Fanuc_WarehouseHandshake
GET
WareHouseClampA_Handshake := _DO1;
END_GET
SET
// Outside -> FB 
_DO1 := WareHouseClampA_Handshake;
END_SET
END_PROPERTY

PROPERTY WareHouseClampB_Handshake : ST_Fanuc_WarehouseHandshake
GET
WareHouseClampB_Handshake := _DO2;
END_GET
SET
// Outside -> FB 
_DO2 := WareHouseClampB_Handshake;
END_SET
END_PROPERTY

PROPERTY Write_OffsetP : INT
SET
_DI11 := Write_OffsetP;
END_SET
END_PROPERTY

PROPERTY Write_OffsetR : INT
SET
_DO12 := Write_OffsetR;
END_SET
END_PROPERTY

PROPERTY Write_OffsetW : INT
SET
_DO10 := Write_OffsetW;
END_SET
END_PROPERTY

PROPERTY Write_OffsetX : INT
SET
_DO7 := Write_OffsetX;
END_SET
END_PROPERTY

PROPERTY Write_OffsetY : INT
SET
_DO8 := Write_OffsetY;
END_SET
END_PROPERTY

PROPERTY Write_OffsetZ : INT
SET
_DO9 := Write_OffsetZ;
END_SET
END_PROPERTY

PROPERTY WriteDataCommand : bool;
SET
_DO6.WritePara_Execute := WriteDataCommand;
END_SET
END_PROPERTY

END_FUNCTION_BLOCK

(* stored: Version 1.1.0.1, ProductVersion 3.1.4024.13
   POU FB_FanucRobot_Basic: Id {0bc73820-43cc-40a7-97c4-2fab14cccb51}, SpecialFunc None
   Folder Action: Id {edf7d6e3-9a68-4529-b8bc-2cf8283228bd}
   Folder HandShake: Id {34c6738e-d1c9-4564-af41-94ad237f911b}
   Folder Method: Id {bbba280c-21c3-4e7b-8832-222384399108}
   Folder ManualService: Id {64fcd5b4-b6c0-410a-99fc-7b04ec43bfda}
   Folder ModeControl: Id {e0884097-7a47-47a4-8710-d105eba518cc}
   Folder MoveBoxToFeedInConveyor: Id {d24354c8-0752-4247-8227-0c4c628ad360}
   Folder MoveBoxToRoundBelt: Id {a64cf708-129e-45dc-9c20-6b863e865e55}
   Folder PulloutConveyor PickupBox: Id {4f0dc620-233f-4dad-8523-fbe97d073f5f}
   Folder RobotAbsMove: Id {a14f3840-2059-4695-b119-5e890098ed13}
   Folder RobotAction: Id {25c36e03-c04a-4cbc-8d24-a38043d60a48}
   Folder Reset: Id {3a33749f-8971-4fa6-9795-0ccd1ed04156}
   Folder Warehouse PickupBox: Id {ec9118d3-dde0-4393-8178-503775ee23a1}
   Folder Warehouse PlaceBox: Id {b7124531-697e-460b-9e24-5f33bf1cd2b0}
   Action A00_BaseUnit: Id {4b81fef1-c7e2-43cd-8410-921d7e0be76d}
   Action A10_ModeControl: Id {0b521170-cd2b-4ae8-b328-da6a70079750}
   Action A20_ErrorHandle: Id {0c94d975-7819-4a36-befd-ccc5ae115868}
   Action A20_StateControl: Id {81cf4bfc-7225-49dc-b241-9fa6442f63f3}
   Property AbsMoveClampA_Handshake: Id {9ca10e9c-f9b4-477a-9222-cf75ee96103c}
   Get Get: Id {dafca030-10f3-4113-bdab-2c49cc0cf766}
   Set Set: Id {beed5ab5-1543-4456-a5e5-4cd33eb0b47e}
   Property AbsMoveClampB_Handshake: Id {01621633-a99e-4779-9806-a9ff51fe7df8}
   Get Get: Id {d7b1afbb-a801-41bb-a33c-a3d73e09d0c7}
   Set Set: Id {d8a60d1c-b211-4de8-820f-240836df59c6}
   Property Bzone_AllowWork: Id {16e5ff50-a1ce-4695-82a6-3ce2c8bd644b}
   Get Get: Id {09d09c79-5a55-4833-b850-4f9560c8f04c}
   Set Set: Id {3fb6f540-fcc6-4366-acb4-c2ee02d5d2f7}
   Property BZoneInWork: Id {5a7a15f1-582a-48c6-a383-b0e0a9ef06e2}
   Get Get: Id {4af81b7b-3e01-4f9d-b3e1-094f83017000}
   Property Command: Id {50b37b0c-06e3-4cd8-b2a3-0609f2429eeb}
   Get Get: Id {07d2c528-3132-463c-8373-acc5f9db2f93}
   Set Set: Id {4d23544e-fb8f-4290-ac34-d2ff3c636e48}
   Method Enable: Id {420d2e98-bc4d-426b-97f0-1e30abfa53b6}
   Method EStop: Id {cc599b02-7c08-4d72-a88e-918e6fea7291}
   Property FanucRobot_MotionStatus: Id {5fae04d8-9d32-4ddf-b0c6-73ff2f6b150c}
   Get Get: Id {9798e90a-130e-48a2-bb3a-44e84ae8232d}
   Method Fault: Id {1ec9f9d0-70ce-406e-976c-dd830579025e}
   Method GetModelState: Id {2bcecda1-4324-45a4-9752-8bf5021a3e42}
   Method GetName: Id {7f258ab7-2346-482c-b77d-d63e1ac3390f}
   Method Hold: Id {670129a5-8c0d-4eba-9348-066e0143afa8}
   Property Homed: Id {365237de-47b6-4ea4-878f-50f0f5a63a15}
   Get Get: Id {da96b359-cd77-4506-9839-ec5f034ff417}
   Property LayerIndex: Id {1ab5a1ea-8c93-4d1b-97c0-85199c8fc151}
   Set Set: Id {2665afd8-a9a8-43ea-8679-80dec21612ba}
   Method M_ActiveRSR01: Id {2fa09742-52c5-44e7-a65c-0e6b6cea633b}
   Method M_ActiveRSR02: Id {6934ebd0-3c5e-4193-aca9-2ebdb53c715c}
   Method M_ActiveRSR03: Id {00f2b2d9-28d8-42e9-add3-77d902dfe5f0}
   Method M_ClearState: Id {c64c69a1-16ce-439b-94a9-5706dddde143}
   Method M_ControlRSR01: Id {feec3cd3-9615-408b-b7d0-dda2b610dc0c}
   Method M_ControlRSR02: Id {236d38d5-eaf6-48b7-a4ff-3f6420cc4238}
   Method M_ControlRSR03: Id {f2e9a683-bc3f-4f9a-a142-0c18d1cb8f51}
   Method M_EnableWith4Input: Id {e0039895-7a35-4336-9f9e-34c531f7ad0d}
   Method M_GetErrorCode: Id {bdd07cb0-8ff7-4210-8ba6-32dfc7c5ec79}
   Method M_Kawasaki_API: Id {e443b7b2-4dca-4f98-8435-0a38e11d4476}
   Method M_ManualService: Id {3bc9292a-ad30-4959-a2aa-bde115855cd0}
   Method M_Reset: Id {acb16e12-1968-4037-ab50-5d2518cf951f}
   Method M_ResetAbsMoveClampACommand: Id {5ac9ab50-da9d-4b03-8910-9e395dc45da3}
   Method M_ResetAbsMoveClampBCommand: Id {779505a1-e0e8-41f4-b118-d278a615c407}
   Method M_ResetAbsMoveCommand: Id {69ddffdb-7ebe-4bc7-bb9f-c57bccbf6080}
   Method M_ResetAllCommand: Id {b1c3f5cb-91f1-4ed6-8126-e8448e0d7725}
   Method M_ResetMoveBoxToFeedInConveyor_ClampA: Id {f310368a-77b5-4326-b5ec-dc54c24761f2}
   Method M_ResetMoveBoxToFeedInConveyor_ClampB: Id {0ddb3060-cc32-49f7-8dcc-368647713061}
   Method M_ResetMoveBoxToFeedInConveyor_ClampBoth: Id {e3330aea-959a-43b0-98fa-a3163b8408c2}
   Method M_ResetMoveBoxToRoundBelt_Both: Id {9739f52a-0108-4485-b7a6-874698275d56}
   Method M_ResetPullOutConveyorPickUpBox_ClampA: Id {bdfc00e6-5f62-4afd-b71c-ba6030407c78}
   Method M_ResetPullOutConveyorPickUpBox_ClampB: Id {90a151a5-87a1-4610-8e85-bf17d6945349}
   Method M_ResetPullOutConveyorPickUpBox_ClampBoth: Id {25692626-124b-4f77-96ee-e2b0f093c492}
   Method M_ResetRobotAbsMove: Id {4711bcbd-34f3-430c-b22d-5704971dc7e7}
   Method M_ResetWareHouseClampACommand: Id {ae8b2728-a591-4e39-9aa5-3d82ff4fec2b}
   Method M_ResetWareHouseClampBCommand: Id {644c5b63-b179-4fb4-8a65-f145752a7ade}
   Method M_ResetWareHouseCommand: Id {2ff0818c-0f30-4019-8bff-66ef399f8a7a}
   Method M_ResetWareHousePickUpBox_ClampA: Id {1aee6a5d-500f-417e-ad1f-3e6964560030}
   Method M_ResetWareHousePickUpBox_ClampB: Id {0621c310-3aa0-40ff-9376-03064c4d014f}
   Method M_ResetWareHousePickUpBox_ClampBoth: Id {c63368a1-12c6-48c9-a934-6ac751358c1d}
   Method M_StartAbsMoveAction_ClampA: Id {83bda59b-1a4e-41f9-b576-9b499ab42d2f}
   Method M_StartAbsMoveAction_ClampB: Id {28b0bbc1-db44-46e5-8f82-74a969153ca1}
   Method M_StartAbsMoveAction_ClampBoth: Id {bf925183-ace6-418c-9cee-8afa2593cf94}
   Method M_StartMoveBoxToFeedInConveyor_ClampA: Id {f4faea24-d129-45d1-b16e-1fd8e64ae554}
   Method M_StartMoveBoxToFeedInConveyor_ClampB: Id {dd9cd97a-41dc-4621-b8d5-5bf601a0cda5}
   Method M_StartMoveBoxToFeedInConveyor_ClampBoth: Id {1a030784-4b78-4b36-863b-175420c701dc}
   Method M_StartMoveBoxToRoundBelt_Both: Id {fec4b46a-488d-4cd5-88fa-6538f533023b}
   Method M_StartMoveBoxToRoundBelt_ClampA: Id {0ae1b5db-63ea-4009-a855-550bb9386903}
   Method M_StartMoveBoxToRoundBelt_ClampB: Id {8e7f1f12-40c9-48e7-8a2a-fba58914953a}
   Method M_StartPullOutConveyorPickUpBox_ClampA: Id {23452bd7-17a5-4a72-ac00-5639a8263a95}
   Method M_StartPullOutConveyorPickUpBox_ClampB: Id {71194040-8e7d-409d-99de-bc2f4e31ce79}
   Method M_StartPullOutConveyorPickUpBox_ClampBoth: Id {4403be70-85d6-4b8b-8851-f7e4761ce126}
   Method M_StartRobotAbsMove: Id {01d0c76d-ae36-47b6-b30a-de3f787b2fc4}
   Method M_StartWarehouseMoveAction_ClampA: Id {91ef9d72-a716-486a-be97-f2f650c69e62}
   Method M_StartWarehouseMoveAction_ClampB: Id {b581a0a0-dce0-4e1d-8e63-3cad9901b7ef}
   Method M_StartWarehouseMoveAction_ClampBoth: Id {06654b35-a456-42d7-bd29-3dbe1a684483}
   Method M_StartWareHousePickUpBox_ClampA: Id {7964043e-453f-407d-a468-3089c7359289}
   Method M_StartWareHousePickUpBox_ClampB: Id {9a90291a-dd06-45ce-b537-8ce007e8507e}
   Method M_StartWareHousePickUpBox_ClampBoth: Id {ae936cf7-0ab9-4e56-8dcb-c5f437f20844}
   Method M_StartWareHousePlaceBox_ClampA: Id {baa9108a-3c22-4cda-9bec-c249bd206fa1}
   Method M_StartWareHousePlaceBox_ClampB: Id {8754649d-8eac-451c-b973-ec7827ac7ee2}
   Method M_StartWareHousePlaceUpBox_ClampBoth: Id {bf4557e7-a91e-4323-9a0d-00cc49ca1fba}
   Method M_SwitchRSR3: Id {642ed4c3-893a-4a19-8622-fb11f05ce680}
   Property Read_OffsetP: Id {6c82c916-f8de-4199-a168-3b123d2255e5}
   Get Get: Id {ebf951ac-1eff-45ea-b072-acff8ed9684d}
   Property Read_OffsetR: Id {495d65ab-ee48-4c7a-b14a-74fa531cf81a}
   Get Get: Id {32876a3b-42a2-4490-b9d2-2861d4b242f3}
   Property Read_OffsetW: Id {c48a6332-9f6e-4ca8-8bdd-3d43f2c595a8}
   Get Get: Id {7fbde413-3c85-432a-aa65-77b2b21fccf6}
   Property Read_OffsetX: Id {3fa75ad4-7620-4e22-a5f2-20d397608dc9}
   Get Get: Id {dd728aae-c532-417b-a4e7-e01f8a051f9f}
   Property Read_OffsetY: Id {db288281-118d-4b8c-93ff-dda102d67711}
   Get Get: Id {8cabd7d8-c80e-42a6-aafd-8f67622022b5}
   Property Read_OffsetZ: Id {ae99ddaf-e55a-4667-845f-be985d1ac667}
   Get Get: Id {8d355c78-d4b7-48b3-8dda-9c564f86ea70}
   Property ReadDataCommand: Id {26667675-c994-46e6-b607-575fc2fd9263}
   Set Set: Id {903d9917-bfe1-43c9-938a-a06eaefbd230}
   Property ReadWrite_Address: Id {6781dbe8-7440-47f4-8ad4-6cb582e6c9e0}
   Set Set: Id {48fc2298-67f5-4f26-982e-888572ee3c7d}
   Property ReadWrite_Area: Id {59b7a0f8-d77f-43c1-9805-3b7c68892e6d}
   Set Set: Id {9c99f2c9-bbe5-4e4f-b75a-72ce481f0101}
   Property ReadWrite_ClampA: Id {a085549c-dbda-4f0e-b4c6-349ff7de3a8b}
   Set Set: Id {022a17fb-311e-4194-9386-c1c26a8ae04e}
   Property ReadWrite_ClampB: Id {ca4a3f5e-ab8f-4d1d-b5aa-d7bade883a30}
   Set Set: Id {6b9a9969-361d-4912-9d8d-afda188eb79e}
   Property ReadWrite_WareHouseA: Id {3444376c-951d-4c84-aece-9c879bf06583}
   Set Set: Id {9a96d751-4031-4a87-964a-96692f692dea}
   Property ReadWrite_WareHouseB: Id {88a6669f-0a91-4074-ae24-2e700d01b656}
   Set Set: Id {40cc9460-638a-418f-aed5-c2317f34e49d}
   Property ReadyOperation: Id {f2cbe881-11d1-4795-a61b-68eebe54f4d0}
   Get Get: Id {c68c5366-afde-4388-9495-87d2437bbdbb}
   Property ReadySetParameter: Id {f862e2fe-bbe2-4dd0-80b9-e483656787e2}
   Get Get: Id {55d56927-8aa5-4a63-a523-2dc6f74efd7b}
   Method ReBoot: Id {61006970-ebad-4c36-b02e-4450798c45a5}
   Property SlideIndex: Id {cdad00d4-ce8e-4829-ab69-2733e792eedb}
   Set Set: Id {523e9471-ef2a-4f0f-b5f3-80bb6e2d6f44}
   Property Status: Id {30f44a75-f2be-4442-ab33-b15efe72f134}
   Get Get: Id {02d59f4e-80a6-45d8-8537-253a29f29757}
   Method Update: Id {facd66d4-4e7a-4ba3-b8ac-c5dd4a0db5b3}
   Property VelocityCommand: Id {7f269991-6c0e-4f8f-b3f2-36310ea13def}
   Get Get: Id {76f6ec90-e16d-44df-b3cb-9e172193fc2e}
   Set Set: Id {530cd5e8-f734-4f34-879a-bc7d5d6777e3}
   Property WareHouseClampA_Handshake: Id {7acafaef-a775-4007-b1e5-393c1d083743}
   Get Get: Id {002d8976-1cf0-4f76-a464-af8311239785}
   Set Set: Id {0d4ae280-df5d-43ef-9392-cdf1f87ada74}
   Property WareHouseClampB_Handshake: Id {5bf83a4f-9b49-4f34-b7d8-59b3cd60328c}
   Get Get: Id {3c28d588-97c1-488a-ac97-e5160dcd453d}
   Set Set: Id {39fecafd-4db6-40fa-b3ab-b2ed6d8841e9}
   Property Write_OffsetP: Id {8354ecc8-c8e5-45fb-8cca-6d52ea33bf64}
   Set Set: Id {9a42a582-1639-4bc4-9f2d-6f292ace5219}
   Property Write_OffsetR: Id {28c5ca91-e008-49f9-a3da-18a12db8ea95}
   Set Set: Id {8c8ca735-3026-4eb4-9710-a21e6b5cef2f}
   Property Write_OffsetW: Id {31abdb60-537d-4bcc-8f23-4db3f432d1b6}
   Set Set: Id {fb4e307f-d70b-4cea-bd7b-d7e3561f647b}
   Property Write_OffsetX: Id {06dc96ab-b65c-4509-83a2-b193442eb6af}
   Set Set: Id {8ab374f2-4e6b-4ff9-ab20-aa480e8297bf}
   Property Write_OffsetY: Id {37542f7d-390b-4ea4-9fd3-d5ea18fdfa54}
   Set Set: Id {db3fc99d-277a-45ff-ab92-af2aecca591a}
   Property Write_OffsetZ: Id {420722f9-d69b-43d4-8f9c-e0b3f4626273}
   Set Set: Id {f424e169-7188-4a29-bcdb-49bff48bfe37}
   Property WriteDataCommand: Id {fecce743-2553-4ed7-af40-316767ad0df6}
   Set Set: Id {bfb1ee87-70cc-488f-b6d8-bf0a1a472085} *)
